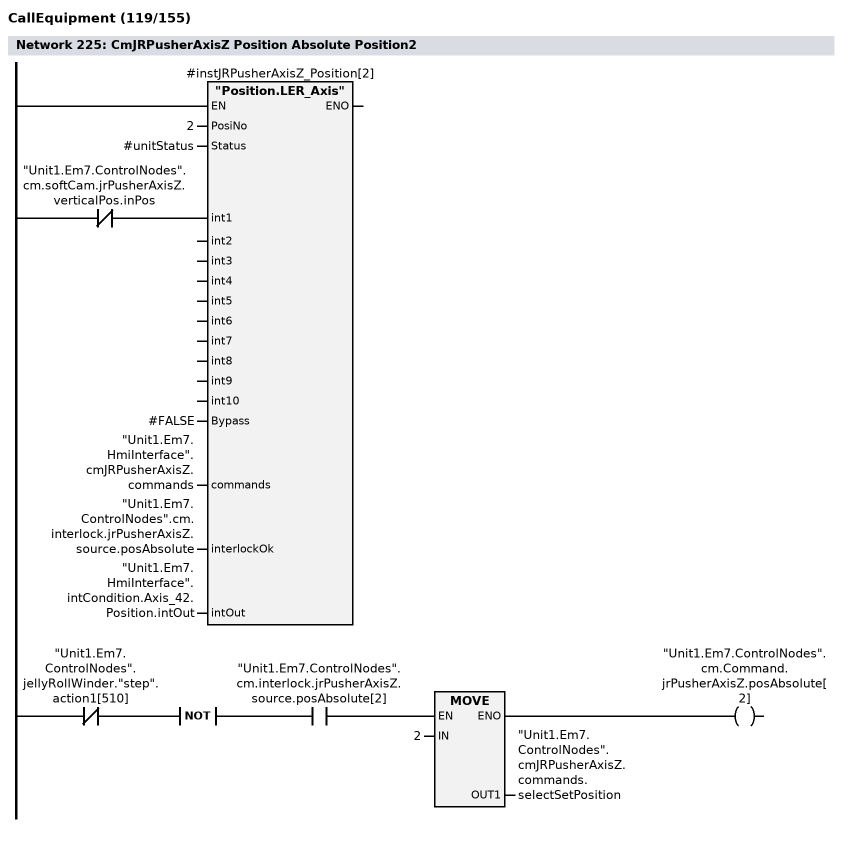
   RUNG wire#powerrail
      #instJRPusherAxisZ_Position[2](int1 := wire#w1, PosiNo := 2, Status := #unitStatus, int2 :=, int3 :=, int4 :=, int5 :=, int6 :=, int7 :=, int8 :=, int9 :=, int10 :=, Bypass := #FALSE, commands := "Unit1.Em7.HmiInterface".cmJRPusherAxisZ.commands, interlockOk := "Unit1.Em7.ControlNodes".cm.interlock.jrPusherAxisZ.source.posAbsolute, intOut := "Unit1.Em7.HmiInterface".intCondition.Axis_42.Position.intOut)
   END_RUNG
   RUNG wire#powerrail
      I_Contact( "Unit1.Em7.ControlNodes".cm.softCam.jrPusherAxisZ.verticalPos.inPos )
   END_RUNG wire#w1
   RUNG wire#powerrail
      I_Contact( "Unit1.Em7.ControlNodes".jellyRollWinder."step".action1[510] )
      Not()
      Contact( "Unit1.Em7.ControlNodes".cm.interlock.jrPusherAxisZ.source.posAbsolute[2] )
      Move(in := 2, out1 => "Unit1.Em7.ControlNodes".cmJRPusherAxisZ.commands.selectSetPosition)
      Coil( "Unit1.Em7.ControlNodes".cm.Command.jrPusherAxisZ.posAbsolute[2] )
   END_RUNG
   // the same network as SCL:
   #instJRPusherAxisZ_Position[2](PosiNo := 2,   // "Position.LER_Axis"
                           Status := #unitStatus,
                           int1 := NOT "Unit1.Em7.ControlNodes".cm.softCam.jrPusherAxisZ.verticalPos.inPos,
                           Bypass := #FALSE,
                           commands := "Unit1.Em7.HmiInterface".cmJRPusherAxisZ.commands,
                           interlockOk := "Unit1.Em7.ControlNodes".cm.interlock.jrPusherAxisZ.source.posAbsolute,
                           intOut := "Unit1.Em7.HmiInterface".intCondition.Axis_42.Position.intOut);
   #_w1 := NOT (NOT "Unit1.Em7.ControlNodes".jellyRollWinder."step".action1[510]) AND "Unit1.Em7.ControlNodes".cm.interlock.jrPusherAxisZ.source.posAbsolute[2];
   IF #_w1 THEN "Unit1.Em7.ControlNodes".cmJRPusherAxisZ.commands.selectSetPosition := 2; END_IF;
   "Unit1.Em7.ControlNodes".cm.Command.jrPusherAxisZ.posAbsolute[2] := #_w1;
END_REGION

REGION Network 226: CmJRPusherAxisZ Position Absolute Position3
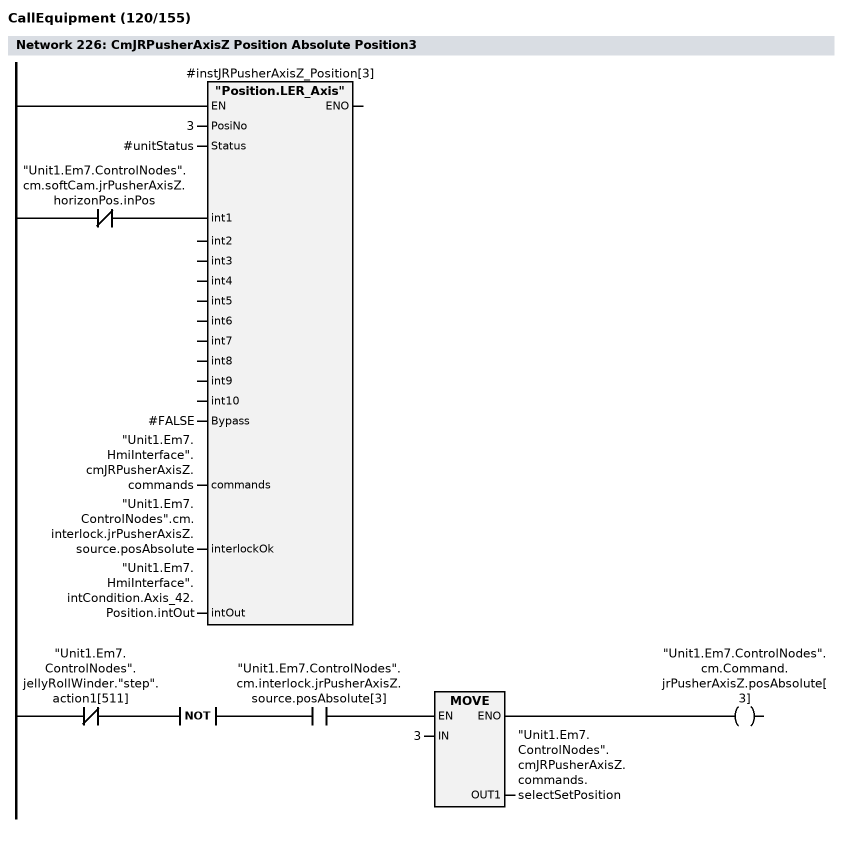
   RUNG wire#powerrail
      #instJRPusherAxisZ_Position[3](int1 := wire#w1, PosiNo := 3, Status := #unitStatus, int2 :=, int3 :=, int4 :=, int5 :=, int6 :=, int7 :=, int8 :=, int9 :=, int10 :=, Bypass := #FALSE, commands := "Unit1.Em7.HmiInterface".cmJRPusherAxisZ.commands, interlockOk := "Unit1.Em7.ControlNodes".cm.interlock.jrPusherAxisZ.source.posAbsolute, intOut := "Unit1.Em7.HmiInterface".intCondition.Axis_42.Position.intOut)
   END_RUNG
   RUNG wire#powerrail
      I_Contact( "Unit1.Em7.ControlNodes".cm.softCam.jrPusherAxisZ.horizonPos.inPos )
   END_RUNG wire#w1
   RUNG wire#powerrail
      I_Contact( "Unit1.Em7.ControlNodes".jellyRollWinder."step".action1[511] )
      Not()
      Contact( "Unit1.Em7.ControlNodes".cm.interlock.jrPusherAxisZ.source.posAbsolute[3] )
      Move(in := 3, out1 => "Unit1.Em7.ControlNodes".cmJRPusherAxisZ.commands.selectSetPosition)
      Coil( "Unit1.Em7.ControlNodes".cm.Command.jrPusherAxisZ.posAbsolute[3] )
   END_RUNG
   // the same network as SCL:
   #instJRPusherAxisZ_Position[3](PosiNo := 3,   // "Position.LER_Axis"
                           Status := #unitStatus,
                           int1 := NOT "Unit1.Em7.ControlNodes".cm.softCam.jrPusherAxisZ.horizonPos.inPos,
                           Bypass := #FALSE,
                           commands := "Unit1.Em7.HmiInterface".cmJRPusherAxisZ.commands,
                           interlockOk := "Unit1.Em7.ControlNodes".cm.interlock.jrPusherAxisZ.source.posAbsolute,
                           intOut := "Unit1.Em7.HmiInterface".intCondition.Axis_42.Position.intOut);
   #_w1 := NOT (NOT "Unit1.Em7.ControlNodes".jellyRollWinder."step".action1[511]) AND "Unit1.Em7.ControlNodes".cm.interlock.jrPusherAxisZ.source.posAbsolute[3];
   IF #_w1 THEN "Unit1.Em7.ControlNodes".cmJRPusherAxisZ.commands.selectSetPosition := 3; END_IF;
   "Unit1.Em7.ControlNodes".cm.Command.jrPusherAxisZ.posAbsolute[3] := #_w1;
END_REGION

REGION Network 227: CmJRPusherAxisZ Position Absolute Position4
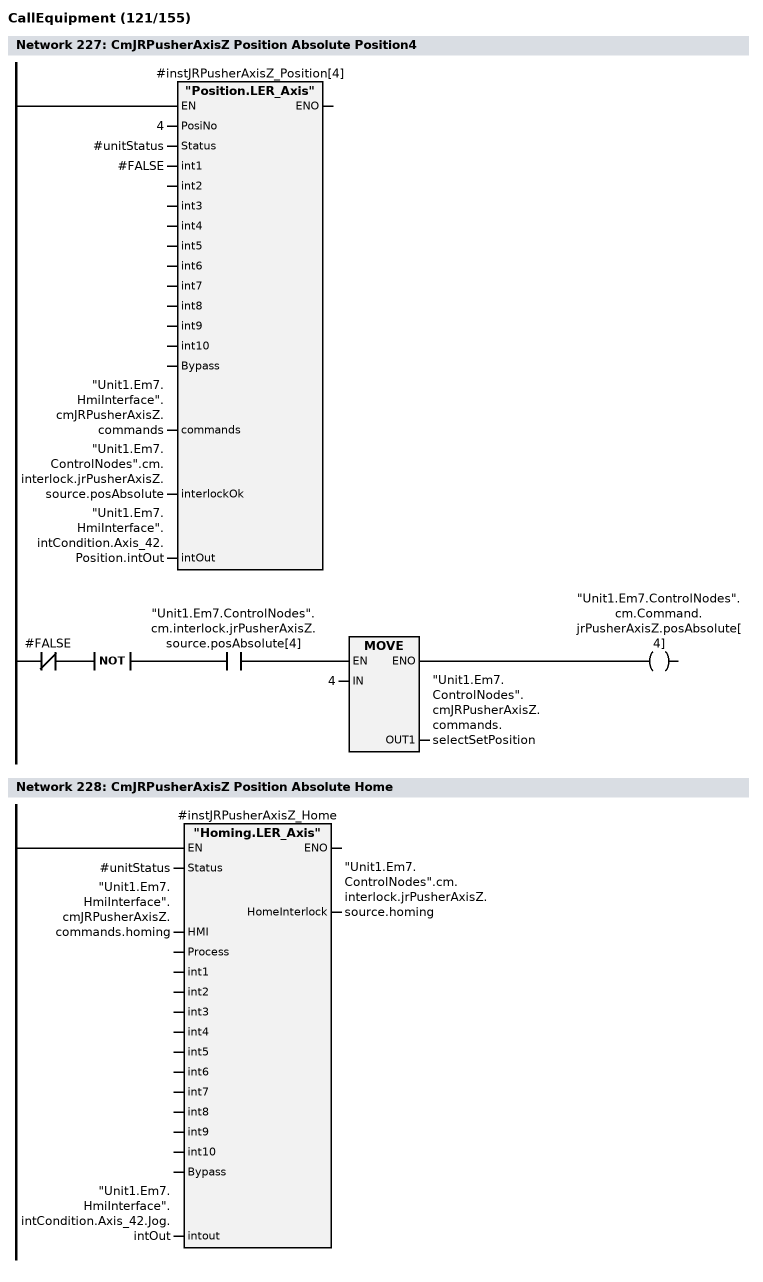
   RUNG wire#powerrail
      #instJRPusherAxisZ_Position[4](PosiNo := 4, Status := #unitStatus, int1 := #FALSE, int2 :=, int3 :=, int4 :=, int5 :=, int6 :=, int7 :=, int8 :=, int9 :=, int10 :=, Bypass :=, commands := "Unit1.Em7.HmiInterface".cmJRPusherAxisZ.commands, interlockOk := "Unit1.Em7.ControlNodes".cm.interlock.jrPusherAxisZ.source.posAbsolute, intOut := "Unit1.Em7.HmiInterface".intCondition.Axis_42.Position.intOut)
   END_RUNG
   RUNG wire#powerrail
      I_Contact( #FALSE )
      Not()
      Contact( "Unit1.Em7.ControlNodes".cm.interlock.jrPusherAxisZ.source.posAbsolute[4] )
      Move(in := 4, out1 => "Unit1.Em7.ControlNodes".cmJRPusherAxisZ.commands.selectSetPosition)
      Coil( "Unit1.Em7.ControlNodes".cm.Command.jrPusherAxisZ.posAbsolute[4] )
   END_RUNG
   // the same network as SCL:
   #instJRPusherAxisZ_Position[4](PosiNo := 4,   // "Position.LER_Axis"
                           Status := #unitStatus,
                           int1 := #FALSE,
                           commands := "Unit1.Em7.HmiInterface".cmJRPusherAxisZ.commands,
                           interlockOk := "Unit1.Em7.ControlNodes".cm.interlock.jrPusherAxisZ.source.posAbsolute,
                           intOut := "Unit1.Em7.HmiInterface".intCondition.Axis_42.Position.intOut);
   #_w1 := NOT (NOT #FALSE) AND "Unit1.Em7.ControlNodes".cm.interlock.jrPusherAxisZ.source.posAbsolute[4];
   IF #_w1 THEN "Unit1.Em7.ControlNodes".cmJRPusherAxisZ.commands.selectSetPosition := 4; END_IF;
   "Unit1.Em7.ControlNodes".cm.Command.jrPusherAxisZ.posAbsolute[4] := #_w1;
END_REGION

REGION Network 228: CmJRPusherAxisZ Position Absolute Home
   RUNG wire#powerrail
      #instJRPusherAxisZ_Home(Status := #unitStatus, HMI := "Unit1.Em7.HmiInterface".cmJRPusherAxisZ.commands.homing, Process :=, int1 :=, int2 :=, int3 :=, int4 :=, int5 :=, int6 :=, int7 :=, int8 :=, int9 :=, int10 :=, Bypass :=, intout := "Unit1.Em7.HmiInterface".intCondition.Axis_42.Jog.intOut, HomeInterlock => "Unit1.Em7.ControlNodes".cm.interlock.jrPusherAxisZ.source.homing)
   END_RUNG
   // the same network as SCL:
   #instJRPusherAxisZ_Home(Status := #unitStatus,   // "Homing.LER_Axis"
                           HMI := "Unit1.Em7.HmiInterface".cmJRPusherAxisZ.commands.homing,
                           intout := "Unit1.Em7.HmiInterface".intCondition.Axis_42.Jog.intOut,
                           HomeInterlock => "Unit1.Em7.ControlNodes".cm.interlock.jrPusherAxisZ.source.homing);
END_REGION

REGION Network 229: CmJRPusherAxisZ Position Absolute Position5
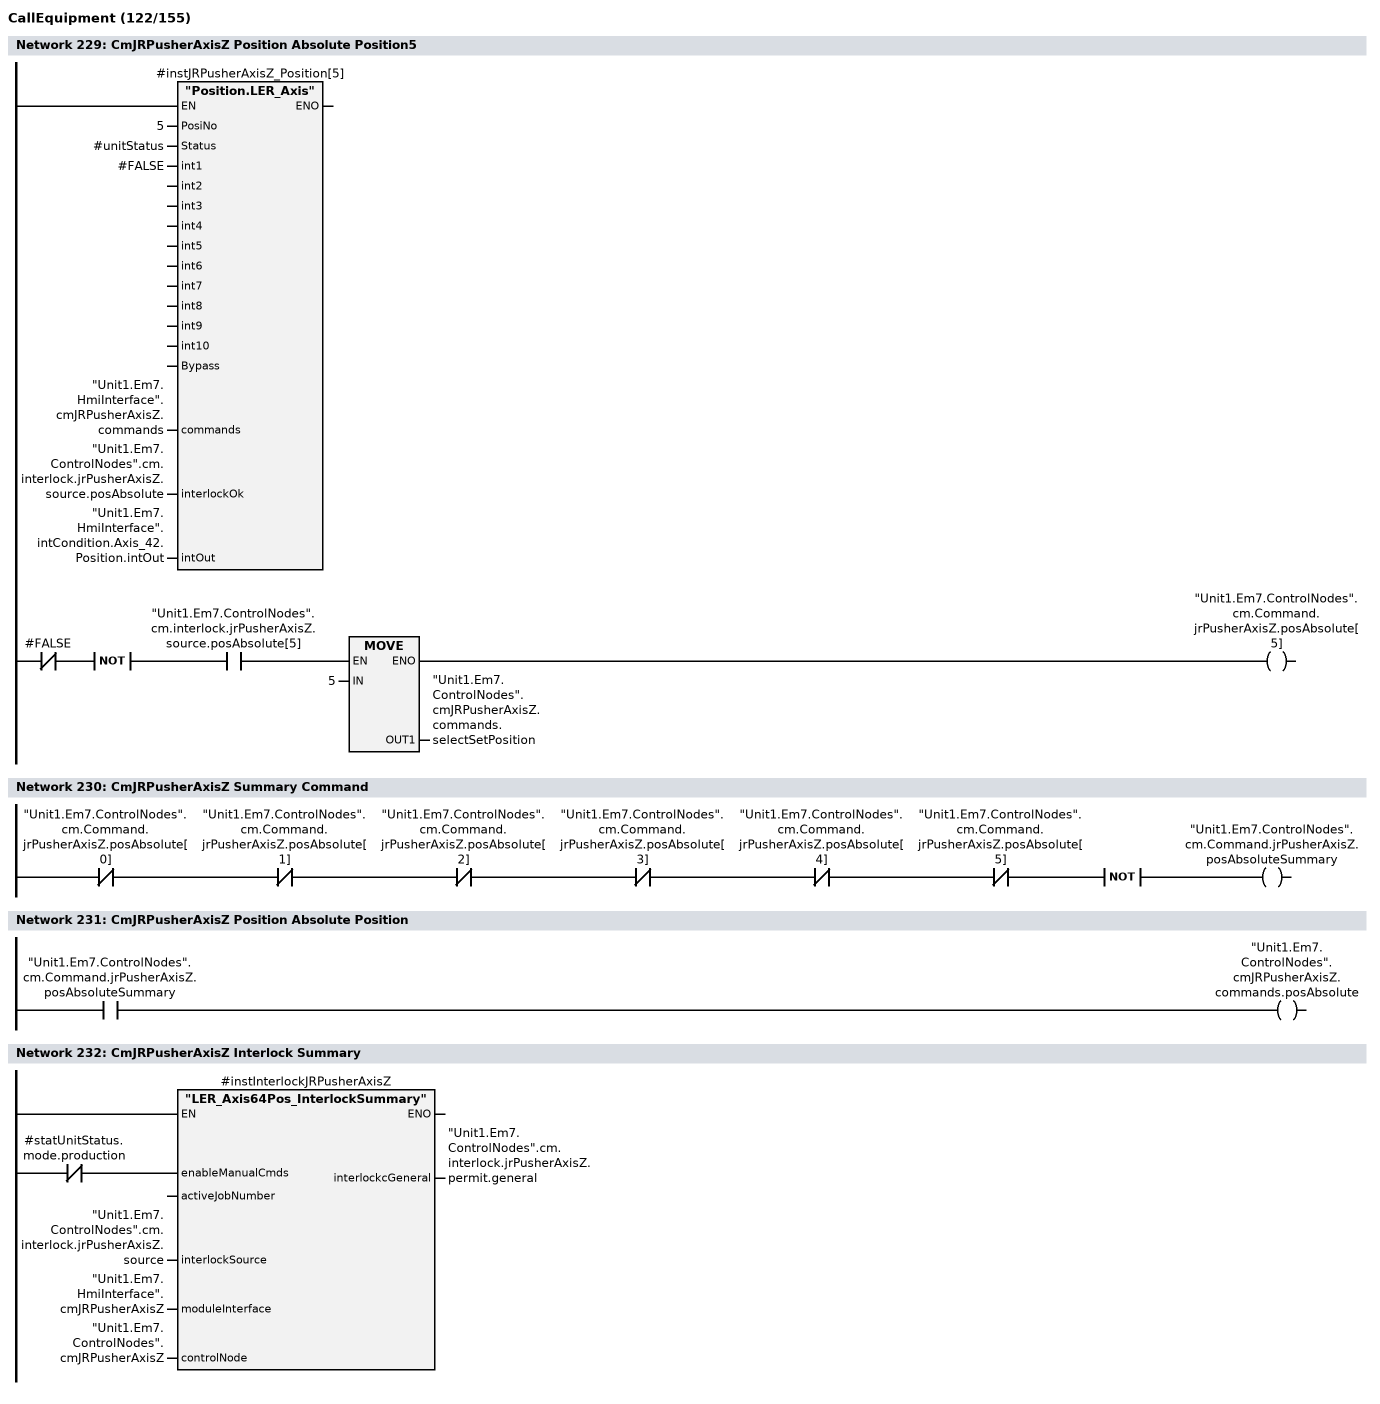
   RUNG wire#powerrail
      #instJRPusherAxisZ_Position[5](PosiNo := 5, Status := #unitStatus, int1 := #FALSE, int2 :=, int3 :=, int4 :=, int5 :=, int6 :=, int7 :=, int8 :=, int9 :=, int10 :=, Bypass :=, commands := "Unit1.Em7.HmiInterface".cmJRPusherAxisZ.commands, interlockOk := "Unit1.Em7.ControlNodes".cm.interlock.jrPusherAxisZ.source.posAbsolute, intOut := "Unit1.Em7.HmiInterface".intCondition.Axis_42.Position.intOut)
   END_RUNG
   RUNG wire#powerrail
      I_Contact( #FALSE )
      Not()
      Contact( "Unit1.Em7.ControlNodes".cm.interlock.jrPusherAxisZ.source.posAbsolute[5] )
      Move(in := 5, out1 => "Unit1.Em7.ControlNodes".cmJRPusherAxisZ.commands.selectSetPosition)
      Coil( "Unit1.Em7.ControlNodes".cm.Command.jrPusherAxisZ.posAbsolute[5] )
   END_RUNG
   // the same network as SCL:
   #instJRPusherAxisZ_Position[5](PosiNo := 5,   // "Position.LER_Axis"
                           Status := #unitStatus,
                           int1 := #FALSE,
                           commands := "Unit1.Em7.HmiInterface".cmJRPusherAxisZ.commands,
                           interlockOk := "Unit1.Em7.ControlNodes".cm.interlock.jrPusherAxisZ.source.posAbsolute,
                           intOut := "Unit1.Em7.HmiInterface".intCondition.Axis_42.Position.intOut);
   #_w1 := NOT (NOT #FALSE) AND "Unit1.Em7.ControlNodes".cm.interlock.jrPusherAxisZ.source.posAbsolute[5];
   IF #_w1 THEN "Unit1.Em7.ControlNodes".cmJRPusherAxisZ.commands.selectSetPosition := 5; END_IF;
   "Unit1.Em7.ControlNodes".cm.Command.jrPusherAxisZ.posAbsolute[5] := #_w1;
END_REGION

REGION Network 230: CmJRPusherAxisZ Summary Command
   RUNG wire#powerrail
      I_Contact( "Unit1.Em7.ControlNodes".cm.Command.jrPusherAxisZ.posAbsolute[0] )
      I_Contact( "Unit1.Em7.ControlNodes".cm.Command.jrPusherAxisZ.posAbsolute[1] )
      I_Contact( "Unit1.Em7.ControlNodes".cm.Command.jrPusherAxisZ.posAbsolute[2] )
      I_Contact( "Unit1.Em7.ControlNodes".cm.Command.jrPusherAxisZ.posAbsolute[3] )
      I_Contact( "Unit1.Em7.ControlNodes".cm.Command.jrPusherAxisZ.posAbsolute[4] )
      I_Contact( "Unit1.Em7.ControlNodes".cm.Command.jrPusherAxisZ.posAbsolute[5] )
      Not()
      Coil( "Unit1.Em7.ControlNodes".cm.Command.jrPusherAxisZ.posAbsoluteSummary )
   END_RUNG
   // the same network as SCL:
   "Unit1.Em7.ControlNodes".cm.Command.jrPusherAxisZ.posAbsoluteSummary := NOT (NOT "Unit1.Em7.ControlNodes".cm.Command.jrPusherAxisZ.posAbsolute[0] AND NOT "Unit1.Em7.ControlNodes".cm.Command.jrPusherAxisZ.posAbsolute[1] AND NOT "Unit1.Em7.ControlNodes".cm.Command.jrPusherAxisZ.posAbsolute[2] AND NOT "Unit1.Em7.ControlNodes".cm.Command.jrPusherAxisZ.posAbsolute[3] AND NOT "Unit1.Em7.ControlNodes".cm.Command.jrPusherAxisZ.posAbsolute[4] AND NOT "Unit1.Em7.ControlNodes".cm.Command.jrPusherAxisZ.posAbsolute[5]);
END_REGION

REGION Network 231: CmJRPusherAxisZ Position Absolute Position
   RUNG wire#powerrail
      Contact( "Unit1.Em7.ControlNodes".cm.Command.jrPusherAxisZ.posAbsoluteSummary )
      Coil( "Unit1.Em7.ControlNodes".cmJRPusherAxisZ.commands.posAbsolute )
   END_RUNG
   // the same network as SCL:
   "Unit1.Em7.ControlNodes".cmJRPusherAxisZ.commands.posAbsolute := "Unit1.Em7.ControlNodes".cm.Command.jrPusherAxisZ.posAbsoluteSummary;
END_REGION

REGION Network 232: CmJRPusherAxisZ Interlock Summary
   RUNG wire#powerrail
      #instInterlockJRPusherAxisZ(enableManualCmds := wire#w1, activeJobNumber :=, interlockSource := "Unit1.Em7.ControlNodes".cm.interlock.jrPusherAxisZ.source, moduleInterface := "Unit1.Em7.HmiInterface".cmJRPusherAxisZ, controlNode := "Unit1.Em7.ControlNodes".cmJRPusherAxisZ, interlockcGeneral => "Unit1.Em7.ControlNodes".cm.interlock.jrPusherAxisZ.permit.general)
   END_RUNG
   RUNG wire#powerrail
      I_Contact( #statUnitStatus.mode.production )
   END_RUNG wire#w1
   // the same network as SCL:
   #instInterlockJRPusherAxisZ(enableManualCmds := NOT #statUnitStatus.mode.production,   // "LER_Axis64Pos_InterlockSummary"
                           interlockSource := "Unit1.Em7.ControlNodes".cm.interlock.jrPusherAxisZ.source,
                           moduleInterface := "Unit1.Em7.HmiInterface".cmJRPusherAxisZ,
                           controlNode := "Unit1.Em7.ControlNodes".cmJRPusherAxisZ,
                           interlockcGeneral => "Unit1.Em7.ControlNodes".cm.interlock.jrPusherAxisZ.permit.general);
END_REGION

REGION Network 233: CmJRPusherAxisZ velocity/speed
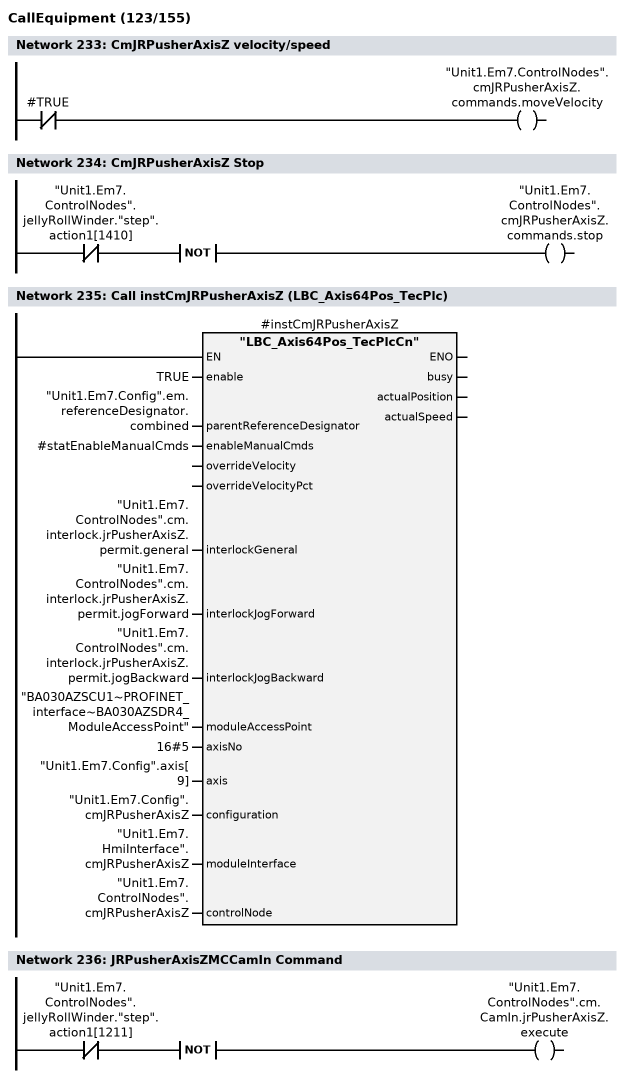
   RUNG wire#powerrail
      I_Contact( #TRUE )
      Coil( "Unit1.Em7.ControlNodes".cmJRPusherAxisZ.commands.moveVelocity )
   END_RUNG
   // the same network as SCL:
   "Unit1.Em7.ControlNodes".cmJRPusherAxisZ.commands.moveVelocity := NOT #TRUE;
END_REGION

REGION Network 234: CmJRPusherAxisZ Stop
   RUNG wire#powerrail
      I_Contact( "Unit1.Em7.ControlNodes".jellyRollWinder."step".action1[1410] )
      Not()
      Coil( "Unit1.Em7.ControlNodes".cmJRPusherAxisZ.commands.stop )
   END_RUNG
   // the same network as SCL:
   "Unit1.Em7.ControlNodes".cmJRPusherAxisZ.commands.stop := NOT (NOT "Unit1.Em7.ControlNodes".jellyRollWinder."step".action1[1410]);
END_REGION

REGION Network 235: Call instCmJRPusherAxisZ (LBC_Axis64Pos_TecPlc)
   RUNG wire#powerrail
      #instCmJRPusherAxisZ(enable := TRUE, parentReferenceDesignator := "Unit1.Em7.Config".em.referenceDesignator.combined, enableManualCmds := #statEnableManualCmds, overrideVelocity :=, overrideVelocityPct :=, interlockGeneral := "Unit1.Em7.ControlNodes".cm.interlock.jrPusherAxisZ.permit.general, interlockJogForward := "Unit1.Em7.ControlNodes".cm.interlock.jrPusherAxisZ.permit.jogForward, interlockJogBackward := "Unit1.Em7.ControlNodes".cm.interlock.jrPusherAxisZ.permit.jogBackward, moduleAccessPoint := "BA030AZSCU1~PROFINET_interface~BA030AZSDR4_ModuleAccessPoint", axisNo := 16#5, axis := "Unit1.Em7.Config".axis[9], configuration := "Unit1.Em7.Config".cmJRPusherAxisZ, moduleInterface := "Unit1.Em7.HmiInterface".cmJRPusherAxisZ, controlNode := "Unit1.Em7.ControlNodes".cmJRPusherAxisZ, busy =>, actualPosition =>, actualSpeed =>)
   END_RUNG
   // the same network as SCL:
   #instCmJRPusherAxisZ(enable := TRUE,   // "LBC_Axis64Pos_TecPlcCn"
                        parentReferenceDesignator := "Unit1.Em7.Config".em.referenceDesignator.combined,
                        enableManualCmds := #statEnableManualCmds,
                        interlockGeneral := "Unit1.Em7.ControlNodes".cm.interlock.jrPusherAxisZ.permit.general,
                        interlockJogForward := "Unit1.Em7.ControlNodes".cm.interlock.jrPusherAxisZ.permit.jogForward,
                        interlockJogBackward := "Unit1.Em7.ControlNodes".cm.interlock.jrPusherAxisZ.permit.jogBackward,
                        moduleAccessPoint := "BA030AZSCU1~PROFINET_interface~BA030AZSDR4_ModuleAccessPoint",
                        axisNo := 16#5,
                        axis := "Unit1.Em7.Config".axis[9],
                        configuration := "Unit1.Em7.Config".cmJRPusherAxisZ,
                        moduleInterface := "Unit1.Em7.HmiInterface".cmJRPusherAxisZ,
                        controlNode := "Unit1.Em7.ControlNodes".cmJRPusherAxisZ);
END_REGION

REGION Network 236: JRPusherAxisZMCCamIn Command
   RUNG wire#powerrail
      I_Contact( "Unit1.Em7.ControlNodes".jellyRollWinder."step".action1[1211] )
      Not()
      Coil( "Unit1.Em7.ControlNodes".cm.CamIn.jrPusherAxisZ.execute )
   END_RUNG
   // the same network as SCL:
   "Unit1.Em7.ControlNodes".cm.CamIn.jrPusherAxisZ.execute := NOT (NOT "Unit1.Em7.ControlNodes".jellyRollWinder."step".action1[1211]);
END_REGION

REGION Network 237: Call instJRPusherAxisZMCCamIn
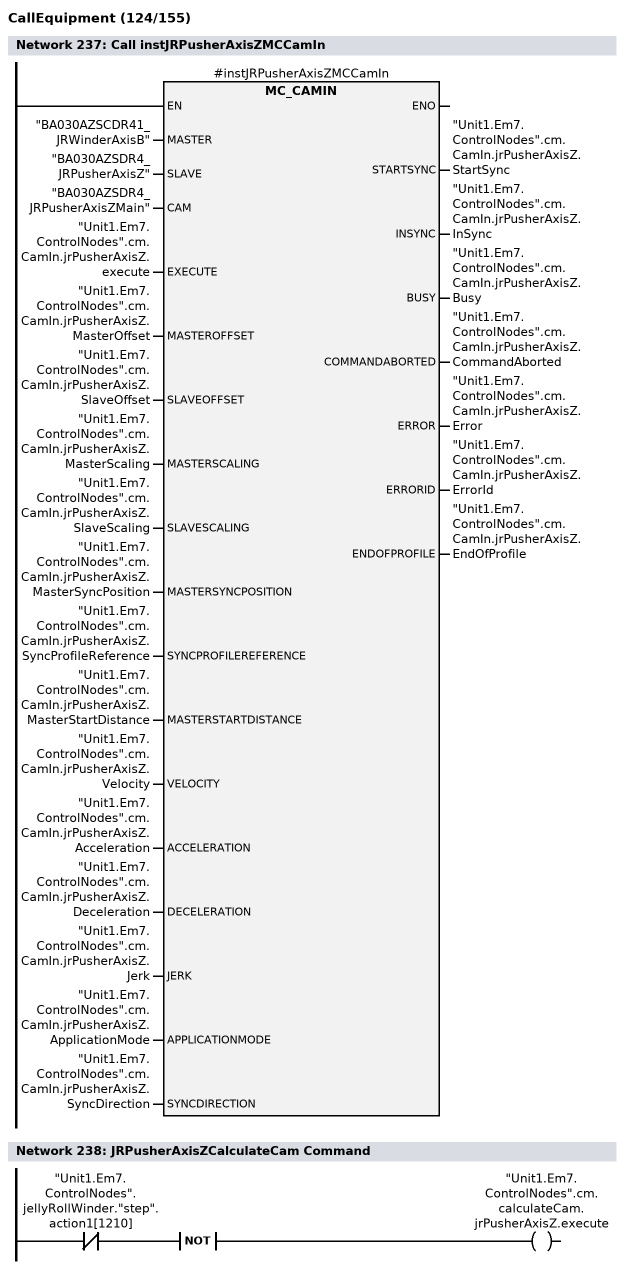
   RUNG wire#powerrail
      #instJRPusherAxisZMCCamIn.MC_CAMIN(Master := "BA030AZSCDR41_JRWinderAxisB", Slave := "BA030AZSDR4_JRPusherAxisZ", Cam := "BA030AZSDR4_JRPusherAxisZMain", Execute := "Unit1.Em7.ControlNodes".cm.CamIn.jrPusherAxisZ.execute, MasterOffset := "Unit1.Em7.ControlNodes".cm.CamIn.jrPusherAxisZ.MasterOffset, SlaveOffset := "Unit1.Em7.ControlNodes".cm.CamIn.jrPusherAxisZ.SlaveOffset, MasterScaling := "Unit1.Em7.ControlNodes".cm.CamIn.jrPusherAxisZ.MasterScaling, SlaveScaling := "Unit1.Em7.ControlNodes".cm.CamIn.jrPusherAxisZ.SlaveScaling, MasterSyncPosition := "Unit1.Em7.ControlNodes".cm.CamIn.jrPusherAxisZ.MasterSyncPosition, SyncProfileReference := "Unit1.Em7.ControlNodes".cm.CamIn.jrPusherAxisZ.SyncProfileReference, MasterStartDistance := "Unit1.Em7.ControlNodes".cm.CamIn.jrPusherAxisZ.MasterStartDistance, Velocity := "Unit1.Em7.ControlNodes".cm.CamIn.jrPusherAxisZ.Velocity, Acceleration := "Unit1.Em7.ControlNodes".cm.CamIn.jrPusherAxisZ.Acceleration, Deceleration := "Unit1.Em7.ControlNodes".cm.CamIn.jrPusherAxisZ.Deceleration, Jerk := "Unit1.Em7.ControlNodes".cm.CamIn.jrPusherAxisZ.Jerk, ApplicationMode := "Unit1.Em7.ControlNodes".cm.CamIn.jrPusherAxisZ.ApplicationMode, SyncDirection := "Unit1.Em7.ControlNodes".cm.CamIn.jrPusherAxisZ.SyncDirection, StartSync => "Unit1.Em7.ControlNodes".cm.CamIn.jrPusherAxisZ.StartSync, InSync => "Unit1.Em7.ControlNodes".cm.CamIn.jrPusherAxisZ.InSync, Busy => "Unit1.Em7.ControlNodes".cm.CamIn.jrPusherAxisZ.Busy, CommandAborted => "Unit1.Em7.ControlNodes".cm.CamIn.jrPusherAxisZ.CommandAborted, Error => "Unit1.Em7.ControlNodes".cm.CamIn.jrPusherAxisZ.Error, ErrorId => "Unit1.Em7.ControlNodes".cm.CamIn.jrPusherAxisZ.ErrorId, EndOfProfile => "Unit1.Em7.ControlNodes".cm.CamIn.jrPusherAxisZ.EndOfProfile)
   END_RUNG
   // the same network as SCL:
   #instJRPusherAxisZMCCamIn(Master := "BA030AZSCDR41_JRWinderAxisB",   // MC_CAMIN
                           Slave := "BA030AZSDR4_JRPusherAxisZ",
                           Cam := "BA030AZSDR4_JRPusherAxisZMain",
                           Execute := "Unit1.Em7.ControlNodes".cm.CamIn.jrPusherAxisZ.execute,
                           MasterOffset := "Unit1.Em7.ControlNodes".cm.CamIn.jrPusherAxisZ.MasterOffset,
                           SlaveOffset := "Unit1.Em7.ControlNodes".cm.CamIn.jrPusherAxisZ.SlaveOffset,
                           MasterScaling := "Unit1.Em7.ControlNodes".cm.CamIn.jrPusherAxisZ.MasterScaling,
                           SlaveScaling := "Unit1.Em7.ControlNodes".cm.CamIn.jrPusherAxisZ.SlaveScaling,
                           MasterSyncPosition := "Unit1.Em7.ControlNodes".cm.CamIn.jrPusherAxisZ.MasterSyncPosition,
                           SyncProfileReference := "Unit1.Em7.ControlNodes".cm.CamIn.jrPusherAxisZ.SyncProfileReference,
                           MasterStartDistance := "Unit1.Em7.ControlNodes".cm.CamIn.jrPusherAxisZ.MasterStartDistance,
                           Velocity := "Unit1.Em7.ControlNodes".cm.CamIn.jrPusherAxisZ.Velocity,
                           Acceleration := "Unit1.Em7.ControlNodes".cm.CamIn.jrPusherAxisZ.Acceleration,
                           Deceleration := "Unit1.Em7.ControlNodes".cm.CamIn.jrPusherAxisZ.Deceleration,
                           Jerk := "Unit1.Em7.ControlNodes".cm.CamIn.jrPusherAxisZ.Jerk,
                           ApplicationMode := "Unit1.Em7.ControlNodes".cm.CamIn.jrPusherAxisZ.ApplicationMode,
                           SyncDirection := "Unit1.Em7.ControlNodes".cm.CamIn.jrPusherAxisZ.SyncDirection,
                           StartSync => "Unit1.Em7.ControlNodes".cm.CamIn.jrPusherAxisZ.StartSync,
                           InSync => "Unit1.Em7.ControlNodes".cm.CamIn.jrPusherAxisZ.InSync,
                           Busy => "Unit1.Em7.ControlNodes".cm.CamIn.jrPusherAxisZ.Busy,
                           CommandAborted => "Unit1.Em7.ControlNodes".cm.CamIn.jrPusherAxisZ.CommandAborted,
                           Error => "Unit1.Em7.ControlNodes".cm.CamIn.jrPusherAxisZ.Error,
                           ErrorId => "Unit1.Em7.ControlNodes".cm.CamIn.jrPusherAxisZ.ErrorId,
                           EndOfProfile => "Unit1.Em7.ControlNodes".cm.CamIn.jrPusherAxisZ.EndOfProfile);
END_REGION

REGION Network 238: JRPusherAxisZCalculateCam Command
   RUNG wire#powerrail
      I_Contact( "Unit1.Em7.ControlNodes".jellyRollWinder."step".action1[1210] )
      Not()
      Coil( "Unit1.Em7.ControlNodes".cm.calculateCam.jrPusherAxisZ.execute )
   END_RUNG
   // the same network as SCL:
   "Unit1.Em7.ControlNodes".cm.calculateCam.jrPusherAxisZ.execute := NOT (NOT "Unit1.Em7.ControlNodes".jellyRollWinder."step".action1[1210]);
END_REGION

REGION Network 239: Call instJRPusherAxisZCalculateCam
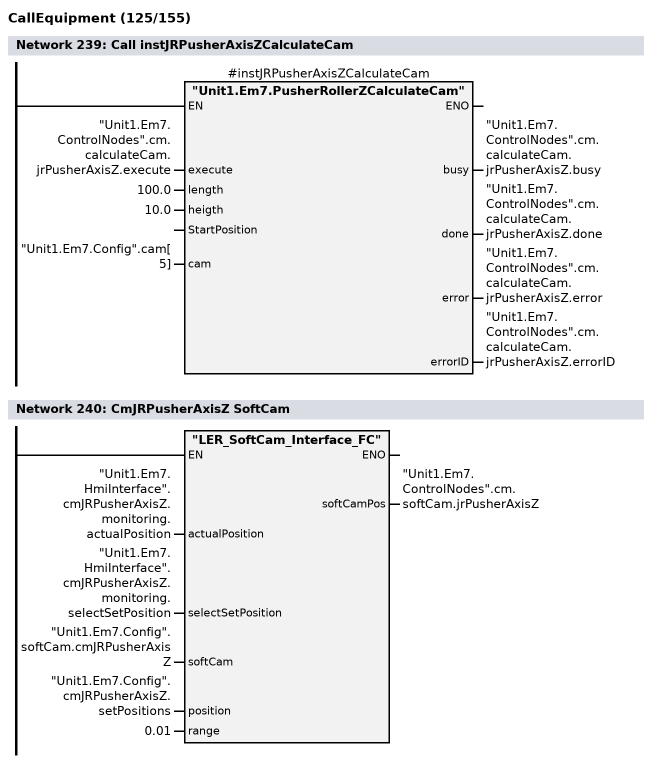
   RUNG wire#powerrail
      #instJRPusherAxisZCalculateCam(execute := "Unit1.Em7.ControlNodes".cm.calculateCam.jrPusherAxisZ.execute, length := 100.0, heigth := 10.0, StartPosition :=, cam := "Unit1.Em7.Config".cam[5], busy => "Unit1.Em7.ControlNodes".cm.calculateCam.jrPusherAxisZ.busy, done => "Unit1.Em7.ControlNodes".cm.calculateCam.jrPusherAxisZ.done, error => "Unit1.Em7.ControlNodes".cm.calculateCam.jrPusherAxisZ.error, errorID => "Unit1.Em7.ControlNodes".cm.calculateCam.jrPusherAxisZ.errorID)
   END_RUNG
   // the same network as SCL:
   #instJRPusherAxisZCalculateCam(execute := "Unit1.Em7.ControlNodes".cm.calculateCam.jrPusherAxisZ.execute,   // "Unit1.Em7.PusherRollerZCalculateCam"
                           length := 100.0,
                           heigth := 10.0,
                           cam := "Unit1.Em7.Config".cam[5],
                           busy => "Unit1.Em7.ControlNodes".cm.calculateCam.jrPusherAxisZ.busy,
                           done => "Unit1.Em7.ControlNodes".cm.calculateCam.jrPusherAxisZ.done,
                           error => "Unit1.Em7.ControlNodes".cm.calculateCam.jrPusherAxisZ.error,
                           errorID => "Unit1.Em7.ControlNodes".cm.calculateCam.jrPusherAxisZ.errorID);
END_REGION

REGION Network 240: CmJRPusherAxisZ SoftCam
   RUNG wire#powerrail
      "LER_SoftCam_Interface_FC"(actualPosition := "Unit1.Em7.HmiInterface".cmJRPusherAxisZ.monitoring.actualPosition, selectSetPosition := "Unit1.Em7.HmiInterface".cmJRPusherAxisZ.monitoring.selectSetPosition, softCam := "Unit1.Em7.Config".softCam.cmJRPusherAxisZ, position := "Unit1.Em7.Config".cmJRPusherAxisZ.setPositions, range := 0.01, softCamPos => "Unit1.Em7.ControlNodes".cm.softCam.jrPusherAxisZ)
   END_RUNG
   // the same network as SCL:
   "LER_SoftCam_Interface_FC"(actualPosition := "Unit1.Em7.HmiInterface".cmJRPusherAxisZ.monitoring.actualPosition,
                           selectSetPosition := "Unit1.Em7.HmiInterface".cmJRPusherAxisZ.monitoring.selectSetPosition,
                           softCam := "Unit1.Em7.Config".softCam.cmJRPusherAxisZ,
                           position := "Unit1.Em7.Config".cmJRPusherAxisZ.setPositions,
                           range := 0.01,
                           softCamPos => "Unit1.Em7.ControlNodes".cm.softCam.jrPusherAxisZ);
END_REGION

REGION Network 241: ******************** Brake Test (Axis) ********************
END_REGION

REGION Network 242: Sepa Clamp And Cutter Z-Axis Brake Test
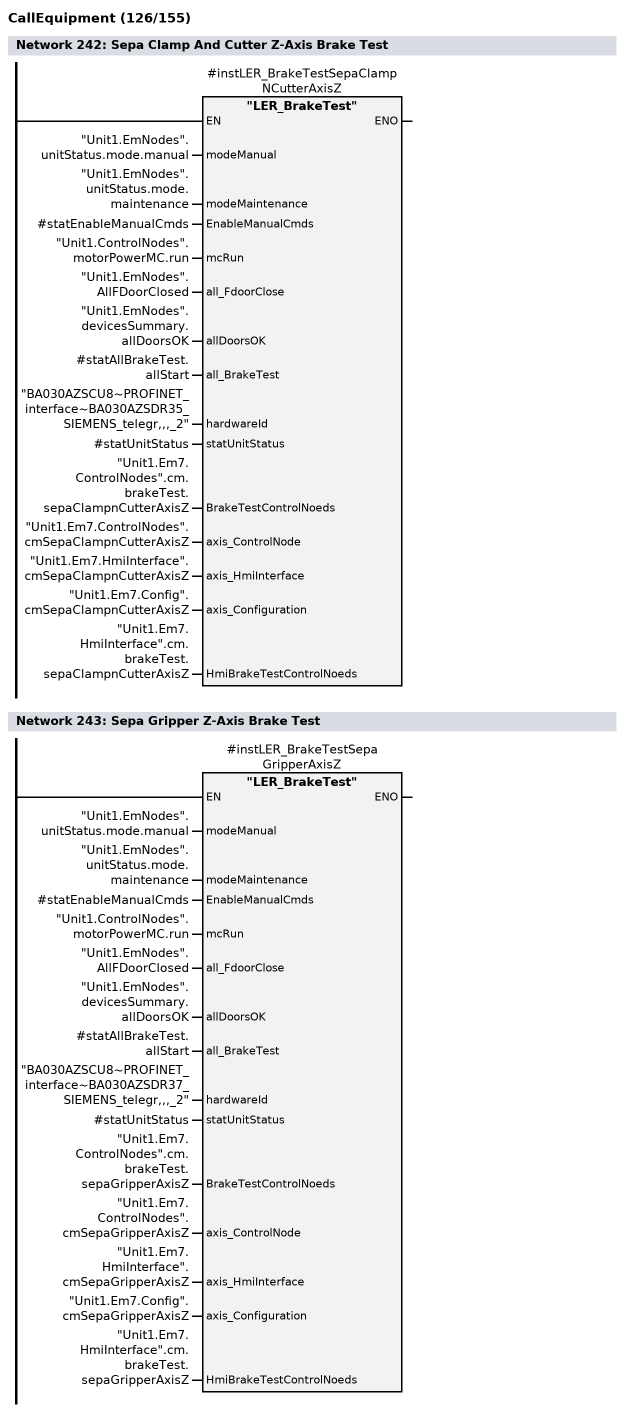
   RUNG wire#powerrail
      #instLER_BrakeTestSepaClampNCutterAxisZ(modeManual := "Unit1.EmNodes".unitStatus.mode.manual, modeMaintenance := "Unit1.EmNodes".unitStatus.mode.maintenance, EnableManualCmds := #statEnableManualCmds, mcRun := "Unit1.ControlNodes".motorPowerMC.run, all_FdoorClose := "Unit1.EmNodes".AllFDoorClosed, allDoorsOK := "Unit1.EmNodes".devicesSummary.allDoorsOK, all_BrakeTest := #statAllBrakeTest.allStart, hardwareId := "BA030AZSCU8~PROFINET_interface~BA030AZSDR35_SIEMENS_telegr,,,_2", statUnitStatus := #statUnitStatus, BrakeTestControlNoeds := "Unit1.Em7.ControlNodes".cm.brakeTest.sepaClampnCutterAxisZ, axis_ControlNode := "Unit1.Em7.ControlNodes".cmSepaClampnCutterAxisZ, axis_HmiInterface := "Unit1.Em7.HmiInterface".cmSepaClampnCutterAxisZ, axis_Configuration := "Unit1.Em7.Config".cmSepaClampnCutterAxisZ, HmiBrakeTestControlNoeds := "Unit1.Em7.HmiInterface".cm.brakeTest.sepaClampnCutterAxisZ)
   END_RUNG
   // the same network as SCL:
   #instLER_BrakeTestSepaClampNCutterAxisZ(modeManual := "Unit1.EmNodes".unitStatus.mode.manual,   // "LER_BrakeTest"
                           modeMaintenance := "Unit1.EmNodes".unitStatus.mode.maintenance,
                           EnableManualCmds := #statEnableManualCmds,
                           mcRun := "Unit1.ControlNodes".motorPowerMC.run,
                           all_FdoorClose := "Unit1.EmNodes".AllFDoorClosed,
                           allDoorsOK := "Unit1.EmNodes".devicesSummary.allDoorsOK,
                           all_BrakeTest := #statAllBrakeTest.allStart,
                           hardwareId := "BA030AZSCU8~PROFINET_interface~BA030AZSDR35_SIEMENS_telegr,,,_2",
                           statUnitStatus := #statUnitStatus,
                           BrakeTestControlNoeds := "Unit1.Em7.ControlNodes".cm.brakeTest.sepaClampnCutterAxisZ,
                           axis_ControlNode := "Unit1.Em7.ControlNodes".cmSepaClampnCutterAxisZ,
                           axis_HmiInterface := "Unit1.Em7.HmiInterface".cmSepaClampnCutterAxisZ,
                           axis_Configuration := "Unit1.Em7.Config".cmSepaClampnCutterAxisZ,
                           HmiBrakeTestControlNoeds := "Unit1.Em7.HmiInterface".cm.brakeTest.sepaClampnCutterAxisZ);
END_REGION

REGION Network 243: Sepa Gripper Z-Axis Brake Test
   RUNG wire#powerrail
      #instLER_BrakeTestSepaGripperAxisZ(modeManual := "Unit1.EmNodes".unitStatus.mode.manual, modeMaintenance := "Unit1.EmNodes".unitStatus.mode.maintenance, EnableManualCmds := #statEnableManualCmds, mcRun := "Unit1.ControlNodes".motorPowerMC.run, all_FdoorClose := "Unit1.EmNodes".AllFDoorClosed, allDoorsOK := "Unit1.EmNodes".devicesSummary.allDoorsOK, all_BrakeTest := #statAllBrakeTest.allStart, hardwareId := "BA030AZSCU8~PROFINET_interface~BA030AZSDR37_SIEMENS_telegr,,,_2", statUnitStatus := #statUnitStatus, BrakeTestControlNoeds := "Unit1.Em7.ControlNodes".cm.brakeTest.sepaGripperAxisZ, axis_ControlNode := "Unit1.Em7.ControlNodes".cmSepaGripperAxisZ, axis_HmiInterface := "Unit1.Em7.HmiInterface".cmSepaGripperAxisZ, axis_Configuration := "Unit1.Em7.Config".cmSepaGripperAxisZ, HmiBrakeTestControlNoeds := "Unit1.Em7.HmiInterface".cm.brakeTest.sepaGripperAxisZ)
   END_RUNG
   // the same network as SCL:
   #instLER_BrakeTestSepaGripperAxisZ(modeManual := "Unit1.EmNodes".unitStatus.mode.manual,   // "LER_BrakeTest"
                           modeMaintenance := "Unit1.EmNodes".unitStatus.mode.maintenance,
                           EnableManualCmds := #statEnableManualCmds,
                           mcRun := "Unit1.ControlNodes".motorPowerMC.run,
                           all_FdoorClose := "Unit1.EmNodes".AllFDoorClosed,
                           allDoorsOK := "Unit1.EmNodes".devicesSummary.allDoorsOK,
                           all_BrakeTest := #statAllBrakeTest.allStart,
                           hardwareId := "BA030AZSCU8~PROFINET_interface~BA030AZSDR37_SIEMENS_telegr,,,_2",
                           statUnitStatus := #statUnitStatus,
                           BrakeTestControlNoeds := "Unit1.Em7.ControlNodes".cm.brakeTest.sepaGripperAxisZ,
                           axis_ControlNode := "Unit1.Em7.ControlNodes".cmSepaGripperAxisZ,
                           axis_HmiInterface := "Unit1.Em7.HmiInterface".cmSepaGripperAxisZ,
                           axis_Configuration := "Unit1.Em7.Config".cmSepaGripperAxisZ,
                           HmiBrakeTestControlNoeds := "Unit1.Em7.HmiInterface".cm.brakeTest.sepaGripperAxisZ);
END_REGION

REGION Network 244: JR Pusher Z-Axis Brake Test
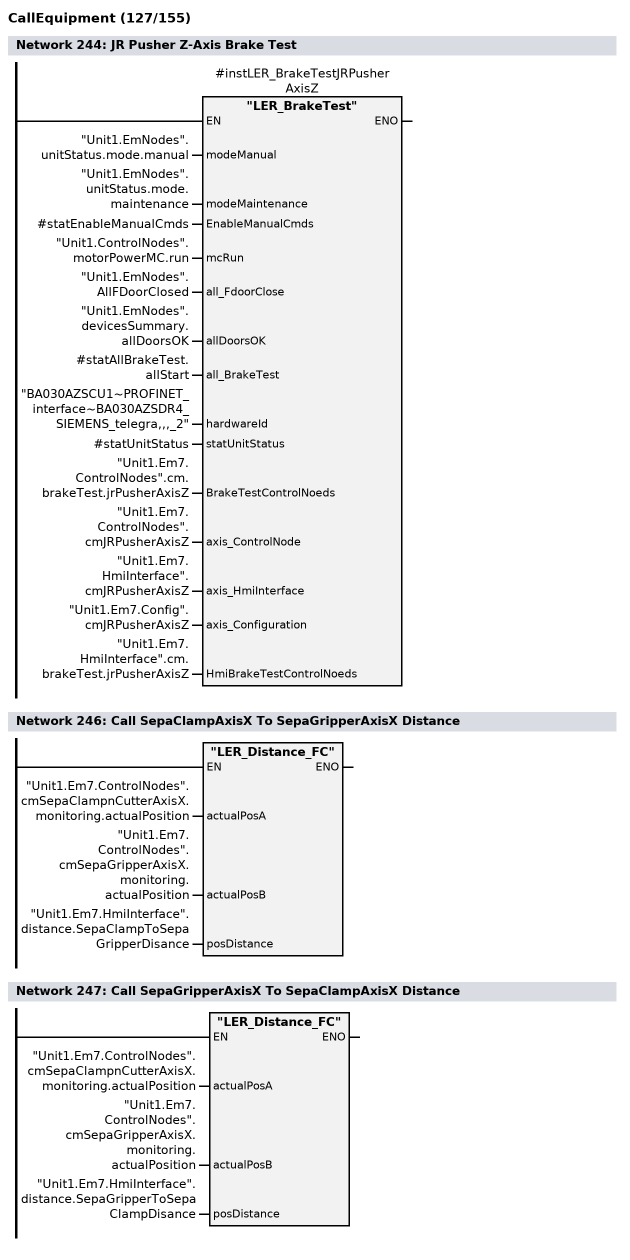
   RUNG wire#powerrail
      #instLER_BrakeTestJRPusherAxisZ(modeManual := "Unit1.EmNodes".unitStatus.mode.manual, modeMaintenance := "Unit1.EmNodes".unitStatus.mode.maintenance, EnableManualCmds := #statEnableManualCmds, mcRun := "Unit1.ControlNodes".motorPowerMC.run, all_FdoorClose := "Unit1.EmNodes".AllFDoorClosed, allDoorsOK := "Unit1.EmNodes".devicesSummary.allDoorsOK, all_BrakeTest := #statAllBrakeTest.allStart, hardwareId := "BA030AZSCU1~PROFINET_interface~BA030AZSDR4_SIEMENS_telegra,,,_2", statUnitStatus := #statUnitStatus, BrakeTestControlNoeds := "Unit1.Em7.ControlNodes".cm.brakeTest.jrPusherAxisZ, axis_ControlNode := "Unit1.Em7.ControlNodes".cmJRPusherAxisZ, axis_HmiInterface := "Unit1.Em7.HmiInterface".cmJRPusherAxisZ, axis_Configuration := "Unit1.Em7.Config".cmJRPusherAxisZ, HmiBrakeTestControlNoeds := "Unit1.Em7.HmiInterface".cm.brakeTest.jrPusherAxisZ)
   END_RUNG
   // the same network as SCL:
   #instLER_BrakeTestJRPusherAxisZ(modeManual := "Unit1.EmNodes".unitStatus.mode.manual,   // "LER_BrakeTest"
                           modeMaintenance := "Unit1.EmNodes".unitStatus.mode.maintenance,
                           EnableManualCmds := #statEnableManualCmds,
                           mcRun := "Unit1.ControlNodes".motorPowerMC.run,
                           all_FdoorClose := "Unit1.EmNodes".AllFDoorClosed,
                           allDoorsOK := "Unit1.EmNodes".devicesSummary.allDoorsOK,
                           all_BrakeTest := #statAllBrakeTest.allStart,
                           hardwareId := "BA030AZSCU1~PROFINET_interface~BA030AZSDR4_SIEMENS_telegra,,,_2",
                           statUnitStatus := #statUnitStatus,
                           BrakeTestControlNoeds := "Unit1.Em7.ControlNodes".cm.brakeTest.jrPusherAxisZ,
                           axis_ControlNode := "Unit1.Em7.ControlNodes".cmJRPusherAxisZ,
                           axis_HmiInterface := "Unit1.Em7.HmiInterface".cmJRPusherAxisZ,
                           axis_Configuration := "Unit1.Em7.Config".cmJRPusherAxisZ,
                           HmiBrakeTestControlNoeds := "Unit1.Em7.HmiInterface".cm.brakeTest.jrPusherAxisZ);
END_REGION

REGION Network 245: ******************** Axis Distance ********************
END_REGION

REGION Network 246: Call SepaClampAxisX To SepaGripperAxisX Distance
   RUNG wire#powerrail
      "LER_Distance_FC"(actualPosA := "Unit1.Em7.ControlNodes".cmSepaClampnCutterAxisX.monitoring.actualPosition, actualPosB := "Unit1.Em7.ControlNodes".cmSepaGripperAxisX.monitoring.actualPosition, posDistance := "Unit1.Em7.HmiInterface".distance.SepaClampToSepaGripperDisance)
   END_RUNG
   // the same network as SCL:
   "LER_Distance_FC"(actualPosA := "Unit1.Em7.ControlNodes".cmSepaClampnCutterAxisX.monitoring.actualPosition,
                     actualPosB := "Unit1.Em7.ControlNodes".cmSepaGripperAxisX.monitoring.actualPosition,
                     posDistance := "Unit1.Em7.HmiInterface".distance.SepaClampToSepaGripperDisance);
END_REGION

REGION Network 247: Call SepaGripperAxisX To SepaClampAxisX Distance
   RUNG wire#powerrail
      "LER_Distance_FC"(actualPosA := "Unit1.Em7.ControlNodes".cmSepaClampnCutterAxisX.monitoring.actualPosition, actualPosB := "Unit1.Em7.ControlNodes".cmSepaGripperAxisX.monitoring.actualPosition, posDistance := "Unit1.Em7.HmiInterface".distance.SepaGripperToSepaClampDisance)
   END_RUNG
   // the same network as SCL:
   "LER_Distance_FC"(actualPosA := "Unit1.Em7.ControlNodes".cmSepaClampnCutterAxisX.monitoring.actualPosition,
                     actualPosB := "Unit1.Em7.ControlNodes".cmSepaGripperAxisX.monitoring.actualPosition,
                     posDistance := "Unit1.Em7.HmiInterface".distance.SepaGripperToSepaClampDisance);
END_REGION

REGION Network 248: ********** Control Modules (TwoWayActuator) **********
END_REGION

REGION Network 249: Reset CMS
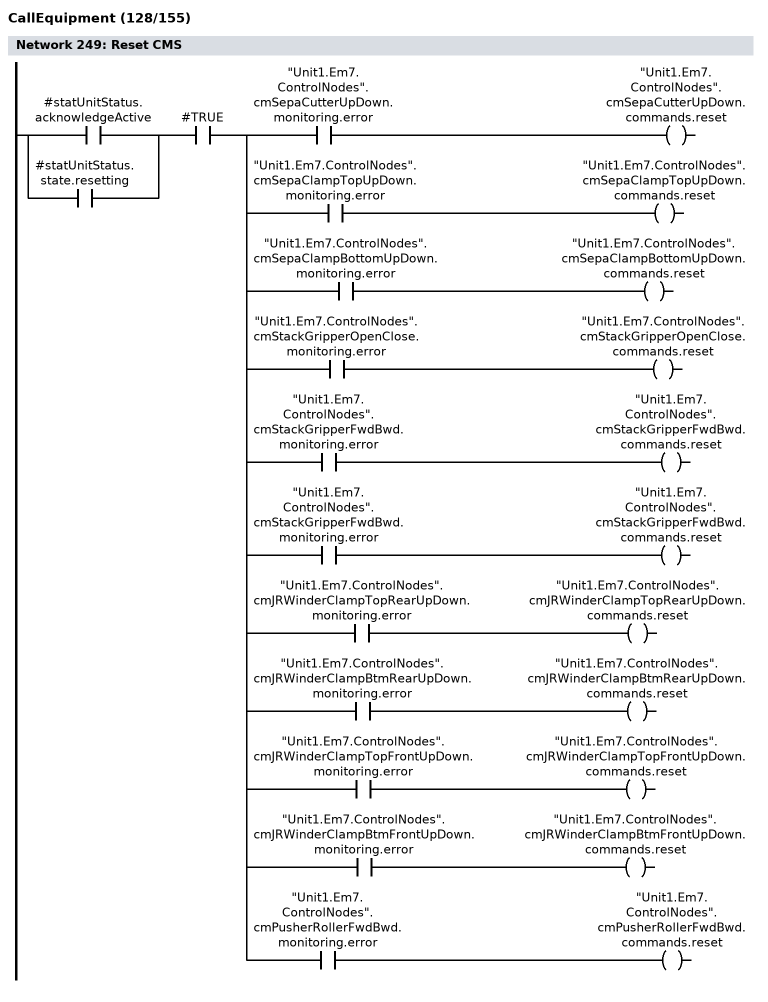
   RUNG wire#powerrail
      Contact( #statUnitStatus.acknowledgeActive )
      wire#w1
      Contact( #TRUE )
      wire#w2
      Contact( "Unit1.Em7.ControlNodes".cmSepaCutterUpDown.monitoring.error )
      Coil( "Unit1.Em7.ControlNodes".cmSepaCutterUpDown.commands.reset )
   END_RUNG
   RUNG wire#powerrail
      Contact( #statUnitStatus.state.resetting )
   END_RUNG wire#w1
   RUNG wire#w2
      Contact( "Unit1.Em7.ControlNodes".cmSepaClampTopUpDown.monitoring.error )
      Coil( "Unit1.Em7.ControlNodes".cmSepaClampTopUpDown.commands.reset )
   END_RUNG
   RUNG wire#w2
      Contact( "Unit1.Em7.ControlNodes".cmSepaClampBottomUpDown.monitoring.error )
      Coil( "Unit1.Em7.ControlNodes".cmSepaClampBottomUpDown.commands.reset )
   END_RUNG
   RUNG wire#w2
      Contact( "Unit1.Em7.ControlNodes".cmStackGripperOpenClose.monitoring.error )
      Coil( "Unit1.Em7.ControlNodes".cmStackGripperOpenClose.commands.reset )
   END_RUNG
   RUNG wire#w2
      Contact( "Unit1.Em7.ControlNodes".cmStackGripperFwdBwd.monitoring.error )
      Coil( "Unit1.Em7.ControlNodes".cmStackGripperFwdBwd.commands.reset )
   END_RUNG
   RUNG wire#w2
      Contact( "Unit1.Em7.ControlNodes".cmStackGripperFwdBwd.monitoring.error )
      Coil( "Unit1.Em7.ControlNodes".cmStackGripperFwdBwd.commands.reset )
   END_RUNG
   RUNG wire#w2
      Contact( "Unit1.Em7.ControlNodes".cmJRWinderClampTopRearUpDown.monitoring.error )
      Coil( "Unit1.Em7.ControlNodes".cmJRWinderClampTopRearUpDown.commands.reset )
   END_RUNG
   RUNG wire#w2
      Contact( "Unit1.Em7.ControlNodes".cmJRWinderClampBtmRearUpDown.monitoring.error )
      Coil( "Unit1.Em7.ControlNodes".cmJRWinderClampBtmRearUpDown.commands.reset )
   END_RUNG
   RUNG wire#w2
      Contact( "Unit1.Em7.ControlNodes".cmJRWinderClampTopFrontUpDown.monitoring.error )
      Coil( "Unit1.Em7.ControlNodes".cmJRWinderClampTopFrontUpDown.commands.reset )
   END_RUNG
   RUNG wire#w2
      Contact( "Unit1.Em7.ControlNodes".cmJRWinderClampBtmFrontUpDown.monitoring.error )
      Coil( "Unit1.Em7.ControlNodes".cmJRWinderClampBtmFrontUpDown.commands.reset )
   END_RUNG
   RUNG wire#w2
      Contact( "Unit1.Em7.ControlNodes".cmPusherRollerFwdBwd.monitoring.error )
      Coil( "Unit1.Em7.ControlNodes".cmPusherRollerFwdBwd.commands.reset )
   END_RUNG
   // the same network as SCL:
   #_w1 := (#statUnitStatus.acknowledgeActive OR #statUnitStatus.state.resetting) AND #TRUE;
   "Unit1.Em7.ControlNodes".cmSepaCutterUpDown.commands.reset := #_w1 AND "Unit1.Em7.ControlNodes".cmSepaCutterUpDown.monitoring.error;
   "Unit1.Em7.ControlNodes".cmSepaClampTopUpDown.commands.reset := #_w1 AND "Unit1.Em7.ControlNodes".cmSepaClampTopUpDown.monitoring.error;
   "Unit1.Em7.ControlNodes".cmSepaClampBottomUpDown.commands.reset := #_w1 AND "Unit1.Em7.ControlNodes".cmSepaClampBottomUpDown.monitoring.error;
   "Unit1.Em7.ControlNodes".cmStackGripperOpenClose.commands.reset := #_w1 AND "Unit1.Em7.ControlNodes".cmStackGripperOpenClose.monitoring.error;
   "Unit1.Em7.ControlNodes".cmStackGripperFwdBwd.commands.reset := #_w1 AND "Unit1.Em7.ControlNodes".cmStackGripperFwdBwd.monitoring.error;
   "Unit1.Em7.ControlNodes".cmStackGripperFwdBwd.commands.reset := #_w1 AND "Unit1.Em7.ControlNodes".cmStackGripperFwdBwd.monitoring.error;
   "Unit1.Em7.ControlNodes".cmJRWinderClampTopRearUpDown.commands.reset := #_w1 AND "Unit1.Em7.ControlNodes".cmJRWinderClampTopRearUpDown.monitoring.error;
   "Unit1.Em7.ControlNodes".cmJRWinderClampBtmRearUpDown.commands.reset := #_w1 AND "Unit1.Em7.ControlNodes".cmJRWinderClampBtmRearUpDown.monitoring.error;
   "Unit1.Em7.ControlNodes".cmJRWinderClampTopFrontUpDown.commands.reset := #_w1 AND "Unit1.Em7.ControlNodes".cmJRWinderClampTopFrontUpDown.monitoring.error;
   "Unit1.Em7.ControlNodes".cmJRWinderClampBtmFrontUpDown.commands.reset := #_w1 AND "Unit1.Em7.ControlNodes".cmJRWinderClampBtmFrontUpDown.monitoring.error;
   "Unit1.Em7.ControlNodes".cmPusherRollerFwdBwd.commands.reset := #_w1 AND "Unit1.Em7.ControlNodes".cmPusherRollerFwdBwd.monitoring.error;
END_REGION

REGION Network 251: CmSepaCutter Up
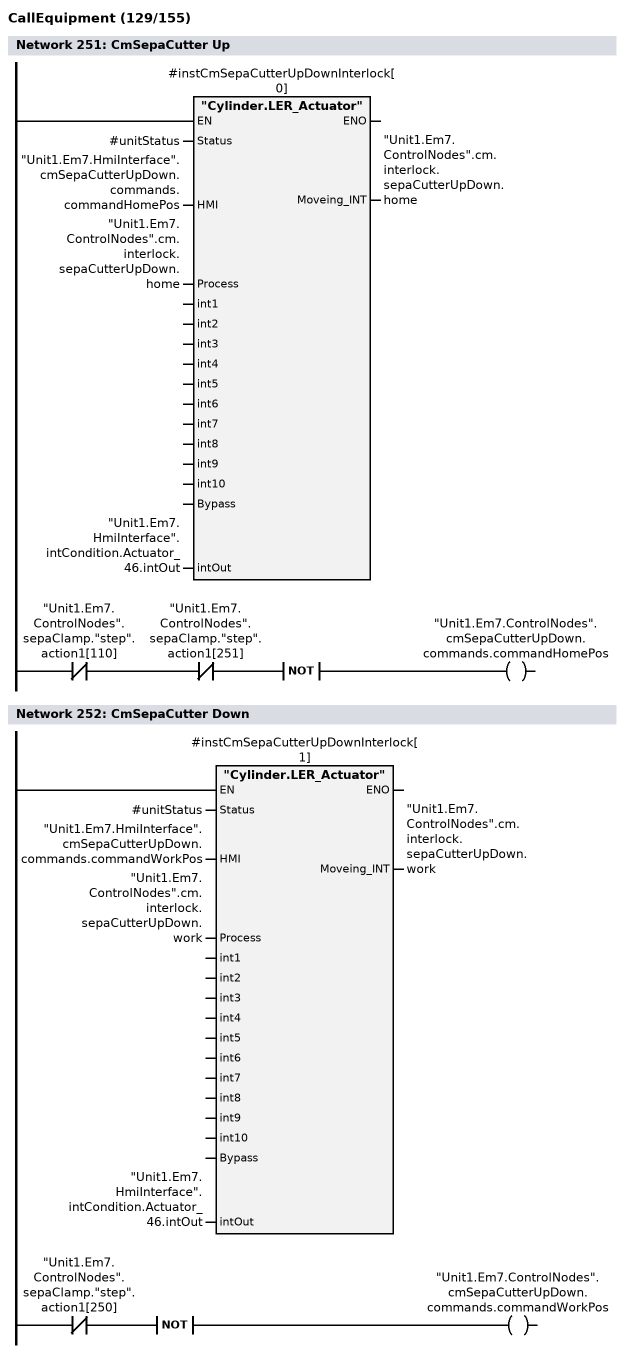
   RUNG wire#powerrail
      #instCmSepaCutterUpDownInterlock[0](Status := #unitStatus, HMI := "Unit1.Em7.HmiInterface".cmSepaCutterUpDown.commands.commandHomePos, Process := "Unit1.Em7.ControlNodes".cm.interlock.sepaCutterUpDown.home, int1 :=, int2 :=, int3 :=, int4 :=, int5 :=, int6 :=, int7 :=, int8 :=, int9 :=, int10 :=, Bypass :=, intOut := "Unit1.Em7.HmiInterface".intCondition.Actuator_46.intOut, Moveing_INT => "Unit1.Em7.ControlNodes".cm.interlock.sepaCutterUpDown.home)
   END_RUNG
   RUNG wire#powerrail
      I_Contact( "Unit1.Em7.ControlNodes".sepaClamp."step".action1[110] )
      I_Contact( "Unit1.Em7.ControlNodes".sepaClamp."step".action1[251] )
      Not()
      Coil( "Unit1.Em7.ControlNodes".cmSepaCutterUpDown.commands.commandHomePos )
   END_RUNG
   // the same network as SCL:
   #instCmSepaCutterUpDownInterlock[0](Status := #unitStatus,   // "Cylinder.LER_Actuator"
                           HMI := "Unit1.Em7.HmiInterface".cmSepaCutterUpDown.commands.commandHomePos,
                           Process := "Unit1.Em7.ControlNodes".cm.interlock.sepaCutterUpDown.home,
                           intOut := "Unit1.Em7.HmiInterface".intCondition.Actuator_46.intOut,
                           Moveing_INT => "Unit1.Em7.ControlNodes".cm.interlock.sepaCutterUpDown.home);
   "Unit1.Em7.ControlNodes".cmSepaCutterUpDown.commands.commandHomePos := NOT (NOT "Unit1.Em7.ControlNodes".sepaClamp."step".action1[110] AND NOT "Unit1.Em7.ControlNodes".sepaClamp."step".action1[251]);
END_REGION

REGION Network 252: CmSepaCutter Down
   RUNG wire#powerrail
      #instCmSepaCutterUpDownInterlock[1](Status := #unitStatus, HMI := "Unit1.Em7.HmiInterface".cmSepaCutterUpDown.commands.commandWorkPos, Process := "Unit1.Em7.ControlNodes".cm.interlock.sepaCutterUpDown.work, int1 :=, int2 :=, int3 :=, int4 :=, int5 :=, int6 :=, int7 :=, int8 :=, int9 :=, int10 :=, Bypass :=, intOut := "Unit1.Em7.HmiInterface".intCondition.Actuator_46.intOut, Moveing_INT => "Unit1.Em7.ControlNodes".cm.interlock.sepaCutterUpDown.work)
   END_RUNG
   RUNG wire#powerrail
      I_Contact( "Unit1.Em7.ControlNodes".sepaClamp."step".action1[250] )
      Not()
      Coil( "Unit1.Em7.ControlNodes".cmSepaCutterUpDown.commands.commandWorkPos )
   END_RUNG
   // the same network as SCL:
   #instCmSepaCutterUpDownInterlock[1](Status := #unitStatus,   // "Cylinder.LER_Actuator"
                           HMI := "Unit1.Em7.HmiInterface".cmSepaCutterUpDown.commands.commandWorkPos,
                           Process := "Unit1.Em7.ControlNodes".cm.interlock.sepaCutterUpDown.work,
                           intOut := "Unit1.Em7.HmiInterface".intCondition.Actuator_46.intOut,
                           Moveing_INT => "Unit1.Em7.ControlNodes".cm.interlock.sepaCutterUpDown.work);
   "Unit1.Em7.ControlNodes".cmSepaCutterUpDown.commands.commandWorkPos := NOT (NOT "Unit1.Em7.ControlNodes".sepaClamp."step".action1[250]);
END_REGION

REGION Network 253: Call instCmSepaCutterUpDown (LBC_TwoWayActuator)
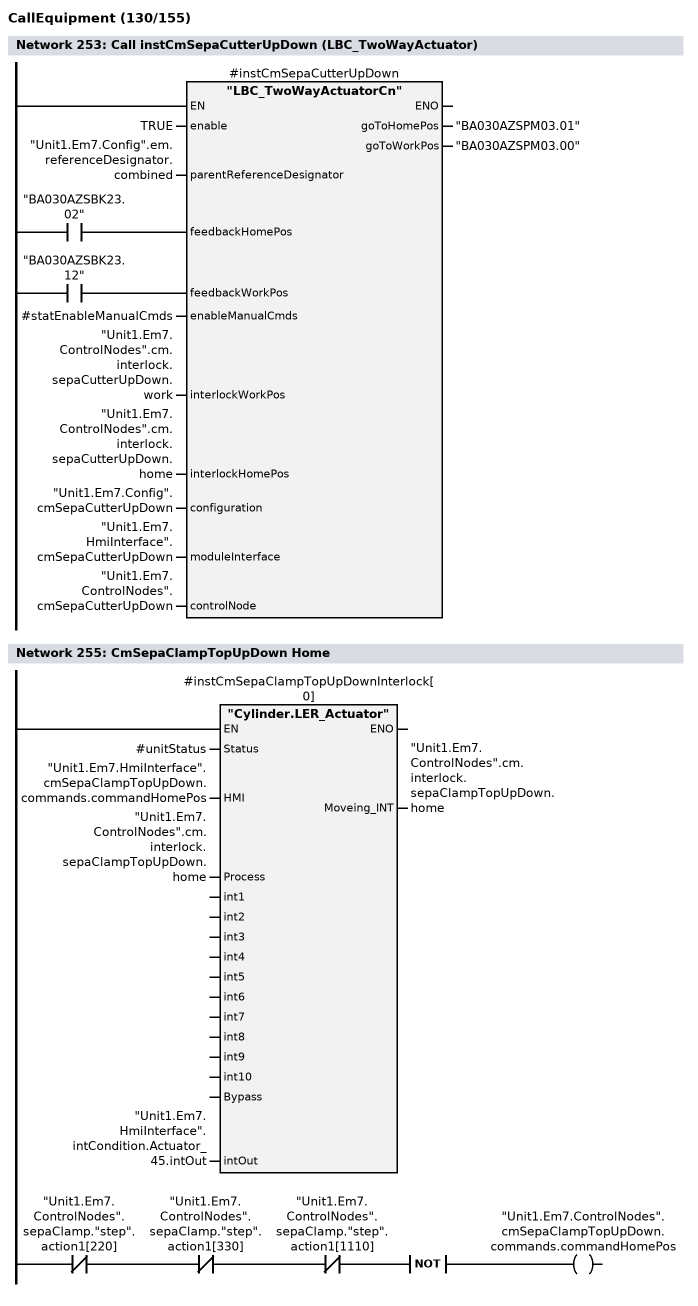
   RUNG wire#powerrail
      #instCmSepaCutterUpDown(feedbackHomePos := wire#w1, feedbackWorkPos := wire#w2, enable := TRUE, parentReferenceDesignator := "Unit1.Em7.Config".em.referenceDesignator.combined, enableManualCmds := #statEnableManualCmds, interlockWorkPos := "Unit1.Em7.ControlNodes".cm.interlock.sepaCutterUpDown.work, interlockHomePos := "Unit1.Em7.ControlNodes".cm.interlock.sepaCutterUpDown.home, configuration := "Unit1.Em7.Config".cmSepaCutterUpDown, moduleInterface := "Unit1.Em7.HmiInterface".cmSepaCutterUpDown, controlNode := "Unit1.Em7.ControlNodes".cmSepaCutterUpDown, goToHomePos => "BA030AZSPM03.01", goToWorkPos => "BA030AZSPM03.00")
   END_RUNG
   RUNG wire#powerrail
      Contact( "BA030AZSBK23.02" )
   END_RUNG wire#w1
   RUNG wire#powerrail
      Contact( "BA030AZSBK23.12" )
   END_RUNG wire#w2
   // the same network as SCL:
   #instCmSepaCutterUpDown(enable := TRUE,   // "LBC_TwoWayActuatorCn"
                           parentReferenceDesignator := "Unit1.Em7.Config".em.referenceDesignator.combined,
                           feedbackHomePos := "BA030AZSBK23.02",
                           feedbackWorkPos := "BA030AZSBK23.12",
                           enableManualCmds := #statEnableManualCmds,
                           interlockWorkPos := "Unit1.Em7.ControlNodes".cm.interlock.sepaCutterUpDown.work,
                           interlockHomePos := "Unit1.Em7.ControlNodes".cm.interlock.sepaCutterUpDown.home,
                           configuration := "Unit1.Em7.Config".cmSepaCutterUpDown,
                           moduleInterface := "Unit1.Em7.HmiInterface".cmSepaCutterUpDown,
                           controlNode := "Unit1.Em7.ControlNodes".cmSepaCutterUpDown,
                           goToHomePos => "BA030AZSPM03.01",
                           goToWorkPos => "BA030AZSPM03.00");
END_REGION

REGION Network 255: CmSepaClampTopUpDown Home
   RUNG wire#powerrail
      #instCmSepaClampTopUpDownInterlock[0](Status := #unitStatus, HMI := "Unit1.Em7.HmiInterface".cmSepaClampTopUpDown.commands.commandHomePos, Process := "Unit1.Em7.ControlNodes".cm.interlock.sepaClampTopUpDown.home, int1 :=, int2 :=, int3 :=, int4 :=, int5 :=, int6 :=, int7 :=, int8 :=, int9 :=, int10 :=, Bypass :=, intOut := "Unit1.Em7.HmiInterface".intCondition.Actuator_45.intOut, Moveing_INT => "Unit1.Em7.ControlNodes".cm.interlock.sepaClampTopUpDown.home)
   END_RUNG
   RUNG wire#powerrail
      I_Contact( "Unit1.Em7.ControlNodes".sepaClamp."step".action1[220] )
      I_Contact( "Unit1.Em7.ControlNodes".sepaClamp."step".action1[330] )
      I_Contact( "Unit1.Em7.ControlNodes".sepaClamp."step".action1[1110] )
      Not()
      Coil( "Unit1.Em7.ControlNodes".cmSepaClampTopUpDown.commands.commandHomePos )
   END_RUNG
   // the same network as SCL:
   #instCmSepaClampTopUpDownInterlock[0](Status := #unitStatus,   // "Cylinder.LER_Actuator"
                           HMI := "Unit1.Em7.HmiInterface".cmSepaClampTopUpDown.commands.commandHomePos,
                           Process := "Unit1.Em7.ControlNodes".cm.interlock.sepaClampTopUpDown.home,
                           intOut := "Unit1.Em7.HmiInterface".intCondition.Actuator_45.intOut,
                           Moveing_INT => "Unit1.Em7.ControlNodes".cm.interlock.sepaClampTopUpDown.home);
   "Unit1.Em7.ControlNodes".cmSepaClampTopUpDown.commands.commandHomePos := NOT (NOT "Unit1.Em7.ControlNodes".sepaClamp."step".action1[220] AND NOT "Unit1.Em7.ControlNodes".sepaClamp."step".action1[330] AND NOT "Unit1.Em7.ControlNodes".sepaClamp."step".action1[1110]);
END_REGION

REGION Network 256: CmSepaClampTopUpDown Work
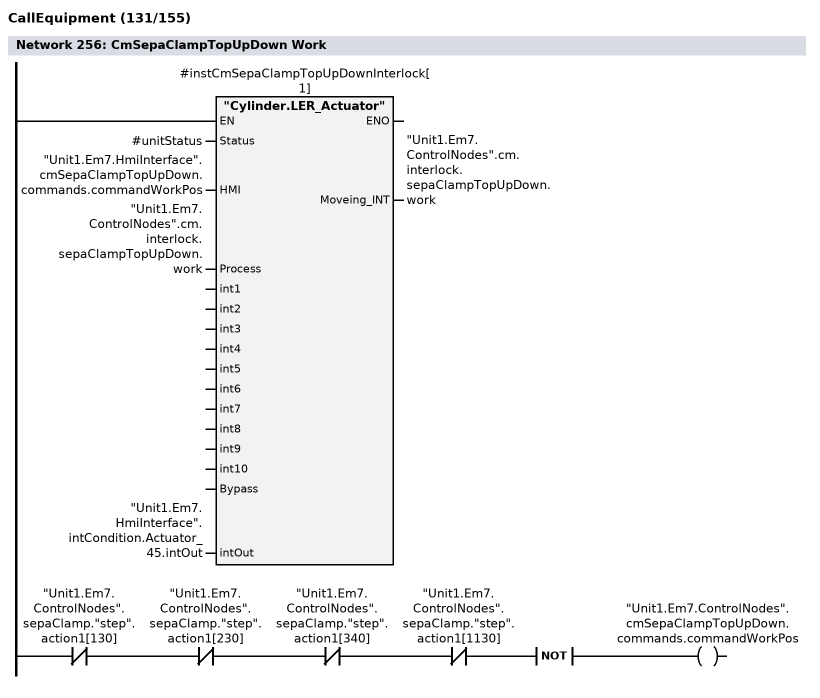
   RUNG wire#powerrail
      #instCmSepaClampTopUpDownInterlock[1](Status := #unitStatus, HMI := "Unit1.Em7.HmiInterface".cmSepaClampTopUpDown.commands.commandWorkPos, Process := "Unit1.Em7.ControlNodes".cm.interlock.sepaClampTopUpDown.work, int1 :=, int2 :=, int3 :=, int4 :=, int5 :=, int6 :=, int7 :=, int8 :=, int9 :=, int10 :=, Bypass :=, intOut := "Unit1.Em7.HmiInterface".intCondition.Actuator_45.intOut, Moveing_INT => "Unit1.Em7.ControlNodes".cm.interlock.sepaClampTopUpDown.work)
   END_RUNG
   RUNG wire#powerrail
      I_Contact( "Unit1.Em7.ControlNodes".sepaClamp."step".action1[130] )
      I_Contact( "Unit1.Em7.ControlNodes".sepaClamp."step".action1[230] )
      I_Contact( "Unit1.Em7.ControlNodes".sepaClamp."step".action1[340] )
      I_Contact( "Unit1.Em7.ControlNodes".sepaClamp."step".action1[1130] )
      Not()
      Coil( "Unit1.Em7.ControlNodes".cmSepaClampTopUpDown.commands.commandWorkPos )
   END_RUNG
   // the same network as SCL:
   #instCmSepaClampTopUpDownInterlock[1](Status := #unitStatus,   // "Cylinder.LER_Actuator"
                           HMI := "Unit1.Em7.HmiInterface".cmSepaClampTopUpDown.commands.commandWorkPos,
                           Process := "Unit1.Em7.ControlNodes".cm.interlock.sepaClampTopUpDown.work,
                           intOut := "Unit1.Em7.HmiInterface".intCondition.Actuator_45.intOut,
                           Moveing_INT => "Unit1.Em7.ControlNodes".cm.interlock.sepaClampTopUpDown.work);
   "Unit1.Em7.ControlNodes".cmSepaClampTopUpDown.commands.commandWorkPos := NOT (NOT "Unit1.Em7.ControlNodes".sepaClamp."step".action1[130] AND NOT "Unit1.Em7.ControlNodes".sepaClamp."step".action1[230] AND NOT "Unit1.Em7.ControlNodes".sepaClamp."step".action1[340] AND NOT "Unit1.Em7.ControlNodes".sepaClamp."step".action1[1130]);
END_REGION

REGION Network 257: Call instCmSepaClampTopUpDown (LBC_TwoWayActuator)
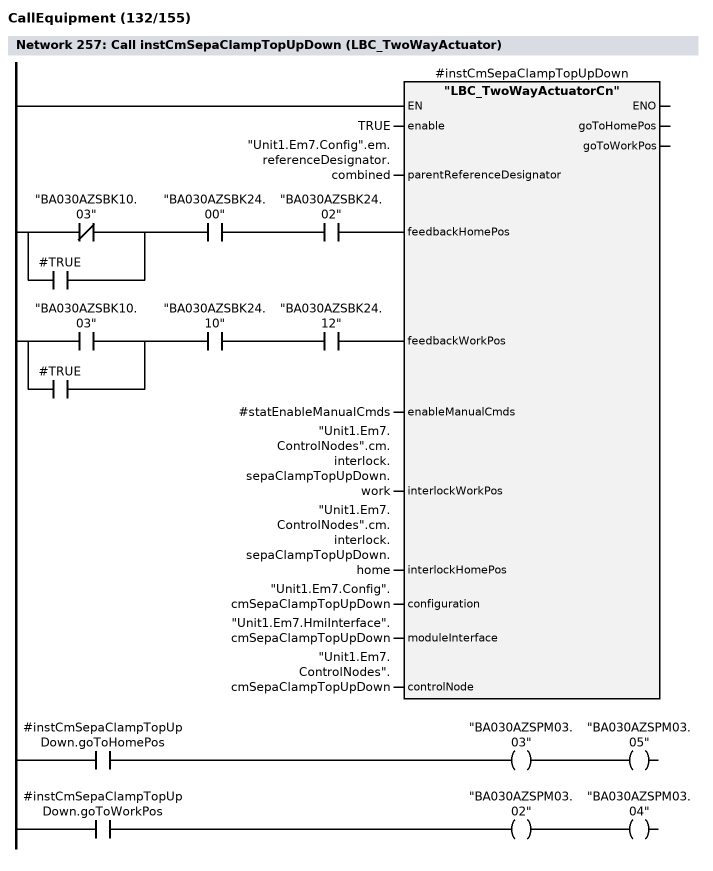
   RUNG wire#powerrail
      #instCmSepaClampTopUpDown(feedbackHomePos := wire#w2, feedbackWorkPos := wire#w4, enable := TRUE, parentReferenceDesignator := "Unit1.Em7.Config".em.referenceDesignator.combined, enableManualCmds := #statEnableManualCmds, interlockWorkPos := "Unit1.Em7.ControlNodes".cm.interlock.sepaClampTopUpDown.work, interlockHomePos := "Unit1.Em7.ControlNodes".cm.interlock.sepaClampTopUpDown.home, configuration := "Unit1.Em7.Config".cmSepaClampTopUpDown, moduleInterface := "Unit1.Em7.HmiInterface".cmSepaClampTopUpDown, controlNode := "Unit1.Em7.ControlNodes".cmSepaClampTopUpDown, goToHomePos =>, goToWorkPos =>)
   END_RUNG
   RUNG wire#powerrail
      I_Contact( "BA030AZSBK10.03" )
      wire#w1
      Contact( "BA030AZSBK24.00" )
      Contact( "BA030AZSBK24.02" )
   END_RUNG wire#w2
   RUNG wire#powerrail
      Contact( #TRUE )
   END_RUNG wire#w1
   RUNG wire#powerrail
      Contact( "BA030AZSBK10.03" )
      wire#w3
      Contact( "BA030AZSBK24.10" )
      Contact( "BA030AZSBK24.12" )
   END_RUNG wire#w4
   RUNG wire#powerrail
      Contact( #TRUE )
   END_RUNG wire#w3
   RUNG wire#powerrail
      Contact( #instCmSepaClampTopUpDown.goToHomePos )
      Coil( "BA030AZSPM03.03" )
      Coil( "BA030AZSPM03.05" )
   END_RUNG
   RUNG wire#powerrail
      Contact( #instCmSepaClampTopUpDown.goToWorkPos )
      Coil( "BA030AZSPM03.02" )
      Coil( "BA030AZSPM03.04" )
   END_RUNG
   // the same network as SCL:
   #instCmSepaClampTopUpDown(enable := TRUE,   // "LBC_TwoWayActuatorCn"
                           parentReferenceDesignator := "Unit1.Em7.Config".em.referenceDesignator.combined,
                           feedbackHomePos := (NOT "BA030AZSBK10.03" OR #TRUE) AND "BA030AZSBK24.00" AND "BA030AZSBK24.02",
                           feedbackWorkPos := ("BA030AZSBK10.03" OR #TRUE) AND "BA030AZSBK24.10" AND "BA030AZSBK24.12",
                           enableManualCmds := #statEnableManualCmds,
                           interlockWorkPos := "Unit1.Em7.ControlNodes".cm.interlock.sepaClampTopUpDown.work,
                           interlockHomePos := "Unit1.Em7.ControlNodes".cm.interlock.sepaClampTopUpDown.home,
                           configuration := "Unit1.Em7.Config".cmSepaClampTopUpDown,
                           moduleInterface := "Unit1.Em7.HmiInterface".cmSepaClampTopUpDown,
                           controlNode := "Unit1.Em7.ControlNodes".cmSepaClampTopUpDown);
   "BA030AZSPM03.03" := #instCmSepaClampTopUpDown.goToHomePos;
   "BA030AZSPM03.05" := #instCmSepaClampTopUpDown.goToHomePos;
   "BA030AZSPM03.02" := #instCmSepaClampTopUpDown.goToWorkPos;
   "BA030AZSPM03.04" := #instCmSepaClampTopUpDown.goToWorkPos;
END_REGION

REGION Network 259: CmSepaClampBottomUpDown Home
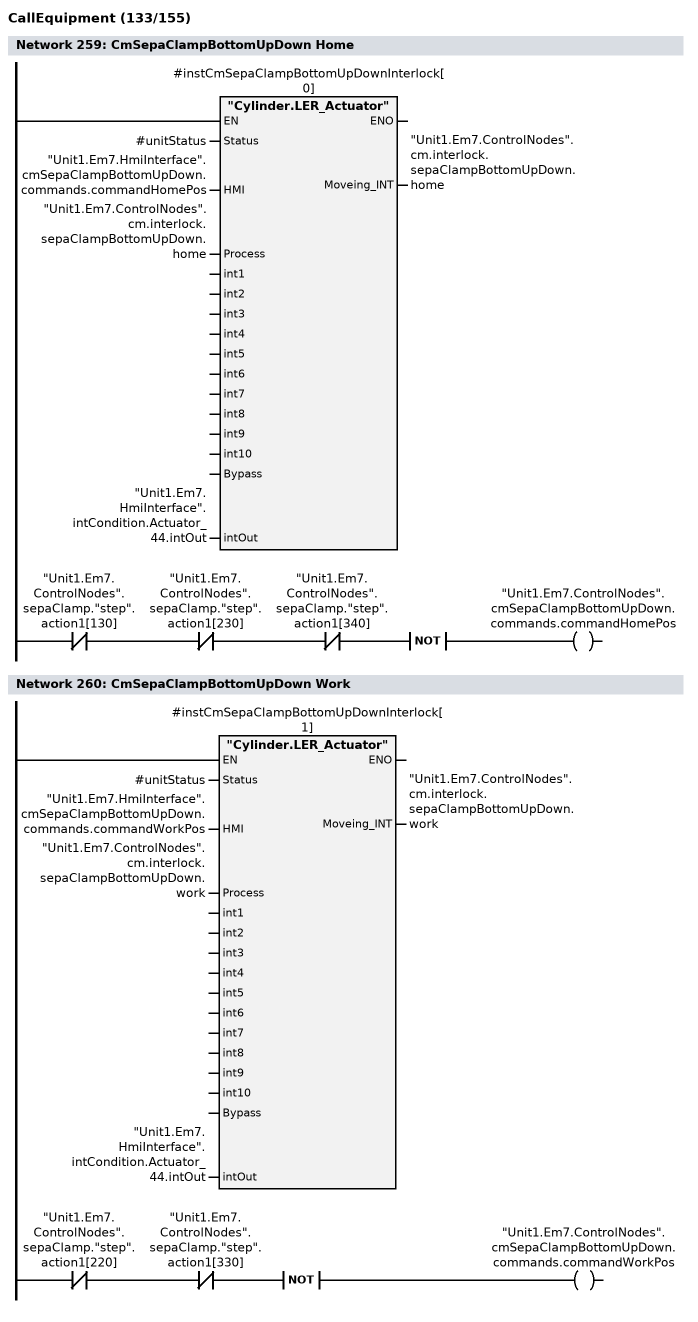
   RUNG wire#powerrail
      #instCmSepaClampBottomUpDownInterlock[0](Status := #unitStatus, HMI := "Unit1.Em7.HmiInterface".cmSepaClampBottomUpDown.commands.commandHomePos, Process := "Unit1.Em7.ControlNodes".cm.interlock.sepaClampBottomUpDown.home, int1 :=, int2 :=, int3 :=, int4 :=, int5 :=, int6 :=, int7 :=, int8 :=, int9 :=, int10 :=, Bypass :=, intOut := "Unit1.Em7.HmiInterface".intCondition.Actuator_44.intOut, Moveing_INT => "Unit1.Em7.ControlNodes".cm.interlock.sepaClampBottomUpDown.home)
   END_RUNG
   RUNG wire#powerrail
      I_Contact( "Unit1.Em7.ControlNodes".sepaClamp."step".action1[130] )
      I_Contact( "Unit1.Em7.ControlNodes".sepaClamp."step".action1[230] )
      I_Contact( "Unit1.Em7.ControlNodes".sepaClamp."step".action1[340] )
      Not()
      Coil( "Unit1.Em7.ControlNodes".cmSepaClampBottomUpDown.commands.commandHomePos )
   END_RUNG
   // the same network as SCL:
   #instCmSepaClampBottomUpDownInterlock[0](Status := #unitStatus,   // "Cylinder.LER_Actuator"
                           HMI := "Unit1.Em7.HmiInterface".cmSepaClampBottomUpDown.commands.commandHomePos,
                           Process := "Unit1.Em7.ControlNodes".cm.interlock.sepaClampBottomUpDown.home,
                           intOut := "Unit1.Em7.HmiInterface".intCondition.Actuator_44.intOut,
                           Moveing_INT => "Unit1.Em7.ControlNodes".cm.interlock.sepaClampBottomUpDown.home);
   "Unit1.Em7.ControlNodes".cmSepaClampBottomUpDown.commands.commandHomePos := NOT (NOT "Unit1.Em7.ControlNodes".sepaClamp."step".action1[130] AND NOT "Unit1.Em7.ControlNodes".sepaClamp."step".action1[230] AND NOT "Unit1.Em7.ControlNodes".sepaClamp."step".action1[340]);
END_REGION

REGION Network 260: CmSepaClampBottomUpDown Work
   RUNG wire#powerrail
      #instCmSepaClampBottomUpDownInterlock[1](Status := #unitStatus, HMI := "Unit1.Em7.HmiInterface".cmSepaClampBottomUpDown.commands.commandWorkPos, Process := "Unit1.Em7.ControlNodes".cm.interlock.sepaClampBottomUpDown.work, int1 :=, int2 :=, int3 :=, int4 :=, int5 :=, int6 :=, int7 :=, int8 :=, int9 :=, int10 :=, Bypass :=, intOut := "Unit1.Em7.HmiInterface".intCondition.Actuator_44.intOut, Moveing_INT => "Unit1.Em7.ControlNodes".cm.interlock.sepaClampBottomUpDown.work)
   END_RUNG
   RUNG wire#powerrail
      I_Contact( "Unit1.Em7.ControlNodes".sepaClamp."step".action1[220] )
      I_Contact( "Unit1.Em7.ControlNodes".sepaClamp."step".action1[330] )
      Not()
      Coil( "Unit1.Em7.ControlNodes".cmSepaClampBottomUpDown.commands.commandWorkPos )
   END_RUNG
   // the same network as SCL:
   #instCmSepaClampBottomUpDownInterlock[1](Status := #unitStatus,   // "Cylinder.LER_Actuator"
                           HMI := "Unit1.Em7.HmiInterface".cmSepaClampBottomUpDown.commands.commandWorkPos,
                           Process := "Unit1.Em7.ControlNodes".cm.interlock.sepaClampBottomUpDown.work,
                           intOut := "Unit1.Em7.HmiInterface".intCondition.Actuator_44.intOut,
                           Moveing_INT => "Unit1.Em7.ControlNodes".cm.interlock.sepaClampBottomUpDown.work);
   "Unit1.Em7.ControlNodes".cmSepaClampBottomUpDown.commands.commandWorkPos := NOT (NOT "Unit1.Em7.ControlNodes".sepaClamp."step".action1[220] AND NOT "Unit1.Em7.ControlNodes".sepaClamp."step".action1[330]);
END_REGION

REGION Network 261: Call instCmSepaClampBottomUpDown (LBC_TwoWayActuator)
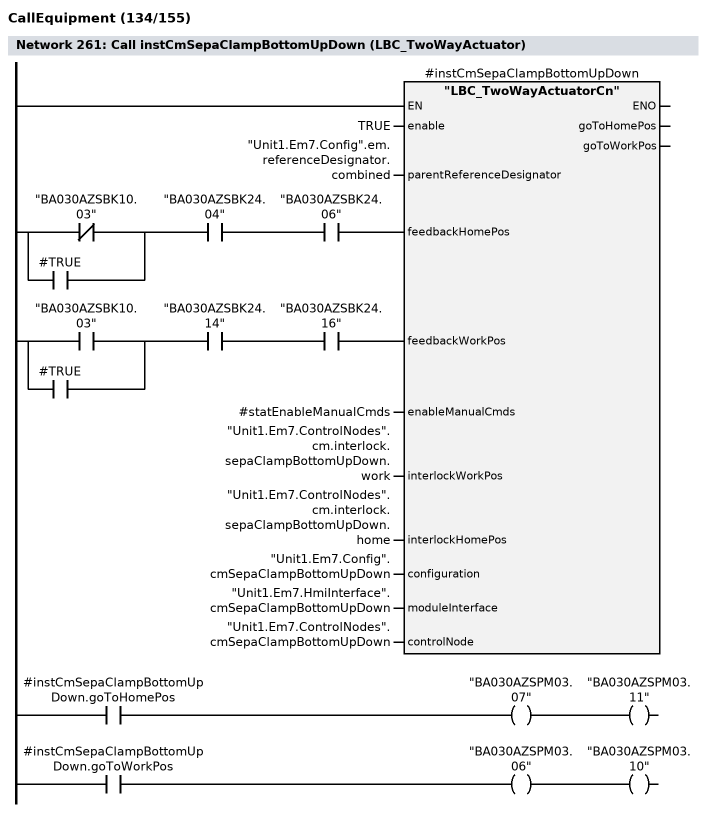
   RUNG wire#powerrail
      #instCmSepaClampBottomUpDown(feedbackHomePos := wire#w2, feedbackWorkPos := wire#w4, enable := TRUE, parentReferenceDesignator := "Unit1.Em7.Config".em.referenceDesignator.combined, enableManualCmds := #statEnableManualCmds, interlockWorkPos := "Unit1.Em7.ControlNodes".cm.interlock.sepaClampBottomUpDown.work, interlockHomePos := "Unit1.Em7.ControlNodes".cm.interlock.sepaClampBottomUpDown.home, configuration := "Unit1.Em7.Config".cmSepaClampBottomUpDown, moduleInterface := "Unit1.Em7.HmiInterface".cmSepaClampBottomUpDown, controlNode := "Unit1.Em7.ControlNodes".cmSepaClampBottomUpDown, goToHomePos =>, goToWorkPos =>)
   END_RUNG
   RUNG wire#powerrail
      I_Contact( "BA030AZSBK10.03" )
      wire#w1
      Contact( "BA030AZSBK24.04" )
      Contact( "BA030AZSBK24.06" )
   END_RUNG wire#w2
   RUNG wire#powerrail
      Contact( #TRUE )
   END_RUNG wire#w1
   RUNG wire#powerrail
      Contact( "BA030AZSBK10.03" )
      wire#w3
      Contact( "BA030AZSBK24.14" )
      Contact( "BA030AZSBK24.16" )
   END_RUNG wire#w4
   RUNG wire#powerrail
      Contact( #TRUE )
   END_RUNG wire#w3
   RUNG wire#powerrail
      Contact( #instCmSepaClampBottomUpDown.goToHomePos )
      Coil( "BA030AZSPM03.07" )
      Coil( "BA030AZSPM03.11" )
   END_RUNG
   RUNG wire#powerrail
      Contact( #instCmSepaClampBottomUpDown.goToWorkPos )
      Coil( "BA030AZSPM03.06" )
      Coil( "BA030AZSPM03.10" )
   END_RUNG
   // the same network as SCL:
   #instCmSepaClampBottomUpDown(enable := TRUE,   // "LBC_TwoWayActuatorCn"
                           parentReferenceDesignator := "Unit1.Em7.Config".em.referenceDesignator.combined,
                           feedbackHomePos := (NOT "BA030AZSBK10.03" OR #TRUE) AND "BA030AZSBK24.04" AND "BA030AZSBK24.06",
                           feedbackWorkPos := ("BA030AZSBK10.03" OR #TRUE) AND "BA030AZSBK24.14" AND "BA030AZSBK24.16",
                           enableManualCmds := #statEnableManualCmds,
                           interlockWorkPos := "Unit1.Em7.ControlNodes".cm.interlock.sepaClampBottomUpDown.work,
                           interlockHomePos := "Unit1.Em7.ControlNodes".cm.interlock.sepaClampBottomUpDown.home,
                           configuration := "Unit1.Em7.Config".cmSepaClampBottomUpDown,
                           moduleInterface := "Unit1.Em7.HmiInterface".cmSepaClampBottomUpDown,
                           controlNode := "Unit1.Em7.ControlNodes".cmSepaClampBottomUpDown);
   "BA030AZSPM03.07" := #instCmSepaClampBottomUpDown.goToHomePos;
   "BA030AZSPM03.11" := #instCmSepaClampBottomUpDown.goToHomePos;
   "BA030AZSPM03.06" := #instCmSepaClampBottomUpDown.goToWorkPos;
   "BA030AZSPM03.10" := #instCmSepaClampBottomUpDown.goToWorkPos;
END_REGION

REGION Network 263: StackGripperOpenClose Home
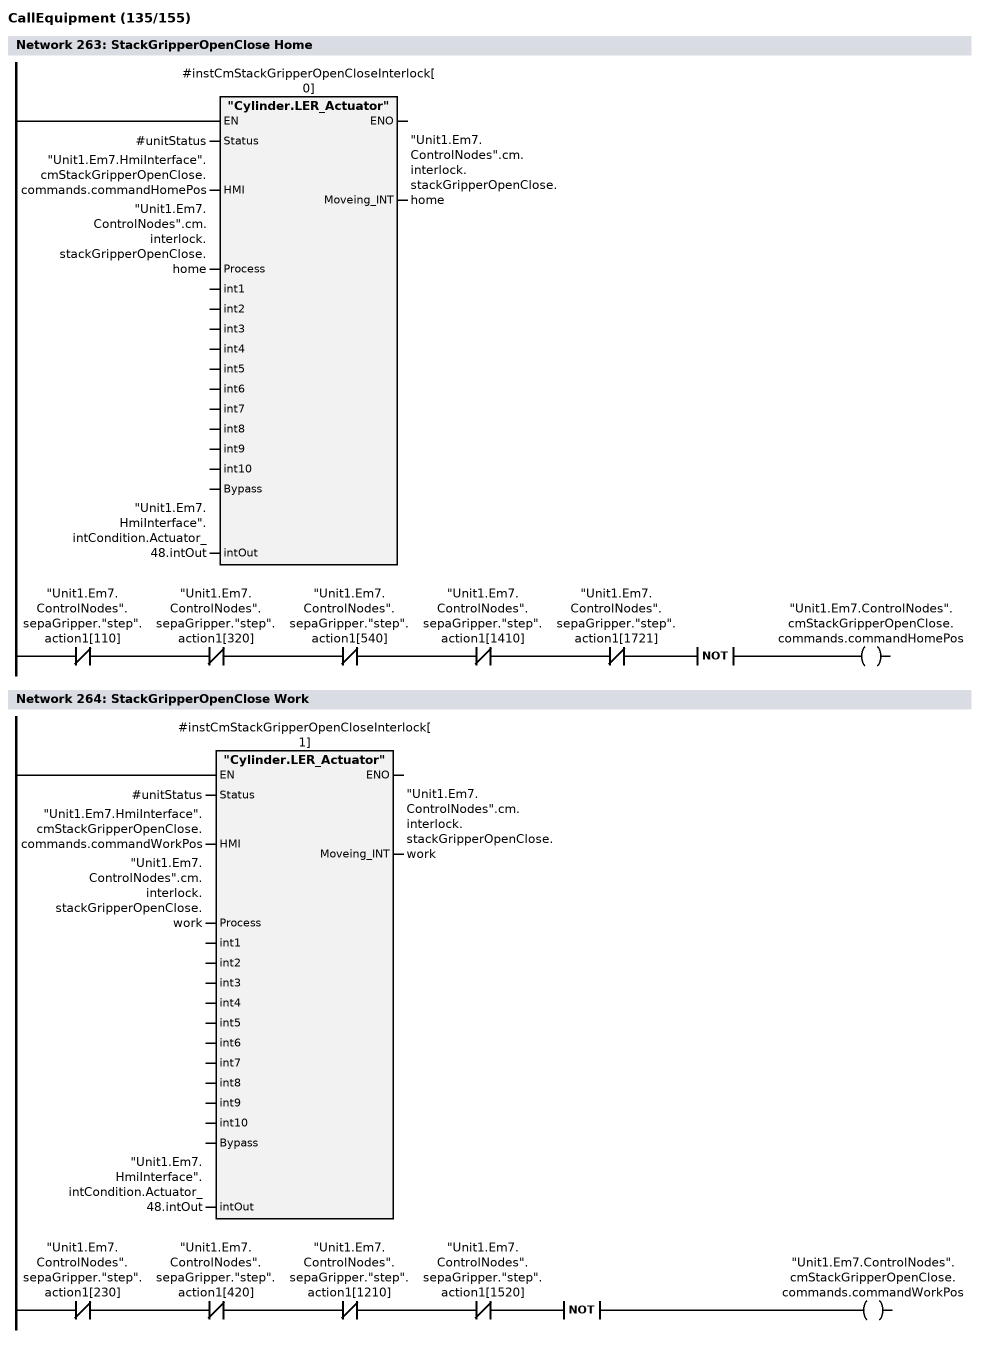
   RUNG wire#powerrail
      #instCmStackGripperOpenCloseInterlock[0](Status := #unitStatus, HMI := "Unit1.Em7.HmiInterface".cmStackGripperOpenClose.commands.commandHomePos, Process := "Unit1.Em7.ControlNodes".cm.interlock.stackGripperOpenClose.home, int1 :=, int2 :=, int3 :=, int4 :=, int5 :=, int6 :=, int7 :=, int8 :=, int9 :=, int10 :=, Bypass :=, intOut := "Unit1.Em7.HmiInterface".intCondition.Actuator_48.intOut, Moveing_INT => "Unit1.Em7.ControlNodes".cm.interlock.stackGripperOpenClose.home)
   END_RUNG
   RUNG wire#powerrail
      I_Contact( "Unit1.Em7.ControlNodes".sepaGripper."step".action1[110] )
      I_Contact( "Unit1.Em7.ControlNodes".sepaGripper."step".action1[320] )
      I_Contact( "Unit1.Em7.ControlNodes".sepaGripper."step".action1[540] )
      I_Contact( "Unit1.Em7.ControlNodes".sepaGripper."step".action1[1410] )
      I_Contact( "Unit1.Em7.ControlNodes".sepaGripper."step".action1[1721] )
      Not()
      Coil( "Unit1.Em7.ControlNodes".cmStackGripperOpenClose.commands.commandHomePos )
   END_RUNG
   // the same network as SCL:
   #instCmStackGripperOpenCloseInterlock[0](Status := #unitStatus,   // "Cylinder.LER_Actuator"
                           HMI := "Unit1.Em7.HmiInterface".cmStackGripperOpenClose.commands.commandHomePos,
                           Process := "Unit1.Em7.ControlNodes".cm.interlock.stackGripperOpenClose.home,
                           intOut := "Unit1.Em7.HmiInterface".intCondition.Actuator_48.intOut,
                           Moveing_INT => "Unit1.Em7.ControlNodes".cm.interlock.stackGripperOpenClose.home);
   "Unit1.Em7.ControlNodes".cmStackGripperOpenClose.commands.commandHomePos := NOT (NOT "Unit1.Em7.ControlNodes".sepaGripper."step".action1[110] AND NOT "Unit1.Em7.ControlNodes".sepaGripper."step".action1[320] AND NOT "Unit1.Em7.ControlNodes".sepaGripper."step".action1[540] AND NOT "Unit1.Em7.ControlNodes".sepaGripper."step".action1[1410] AND NOT "Unit1.Em7.ControlNodes".sepaGripper."step".action1[1721]);
END_REGION

REGION Network 264: StackGripperOpenClose Work
   RUNG wire#powerrail
      #instCmStackGripperOpenCloseInterlock[1](Status := #unitStatus, HMI := "Unit1.Em7.HmiInterface".cmStackGripperOpenClose.commands.commandWorkPos, Process := "Unit1.Em7.ControlNodes".cm.interlock.stackGripperOpenClose.work, int1 :=, int2 :=, int3 :=, int4 :=, int5 :=, int6 :=, int7 :=, int8 :=, int9 :=, int10 :=, Bypass :=, intOut := "Unit1.Em7.HmiInterface".intCondition.Actuator_48.intOut, Moveing_INT => "Unit1.Em7.ControlNodes".cm.interlock.stackGripperOpenClose.work)
   END_RUNG
   RUNG wire#powerrail
      I_Contact( "Unit1.Em7.ControlNodes".sepaGripper."step".action1[230] )
      I_Contact( "Unit1.Em7.ControlNodes".sepaGripper."step".action1[420] )
      I_Contact( "Unit1.Em7.ControlNodes".sepaGripper."step".action1[1210] )
      I_Contact( "Unit1.Em7.ControlNodes".sepaGripper."step".action1[1520] )
      Not()
      Coil( "Unit1.Em7.ControlNodes".cmStackGripperOpenClose.commands.commandWorkPos )
   END_RUNG
   // the same network as SCL:
   #instCmStackGripperOpenCloseInterlock[1](Status := #unitStatus,   // "Cylinder.LER_Actuator"
                           HMI := "Unit1.Em7.HmiInterface".cmStackGripperOpenClose.commands.commandWorkPos,
                           Process := "Unit1.Em7.ControlNodes".cm.interlock.stackGripperOpenClose.work,
                           intOut := "Unit1.Em7.HmiInterface".intCondition.Actuator_48.intOut,
                           Moveing_INT => "Unit1.Em7.ControlNodes".cm.interlock.stackGripperOpenClose.work);
   "Unit1.Em7.ControlNodes".cmStackGripperOpenClose.commands.commandWorkPos := NOT (NOT "Unit1.Em7.ControlNodes".sepaGripper."step".action1[230] AND NOT "Unit1.Em7.ControlNodes".sepaGripper."step".action1[420] AND NOT "Unit1.Em7.ControlNodes".sepaGripper."step".action1[1210] AND NOT "Unit1.Em7.ControlNodes".sepaGripper."step".action1[1520]);
END_REGION

REGION Network 265: Call instCmStackGripperOpenClose (LBC_TwoWayActuator)
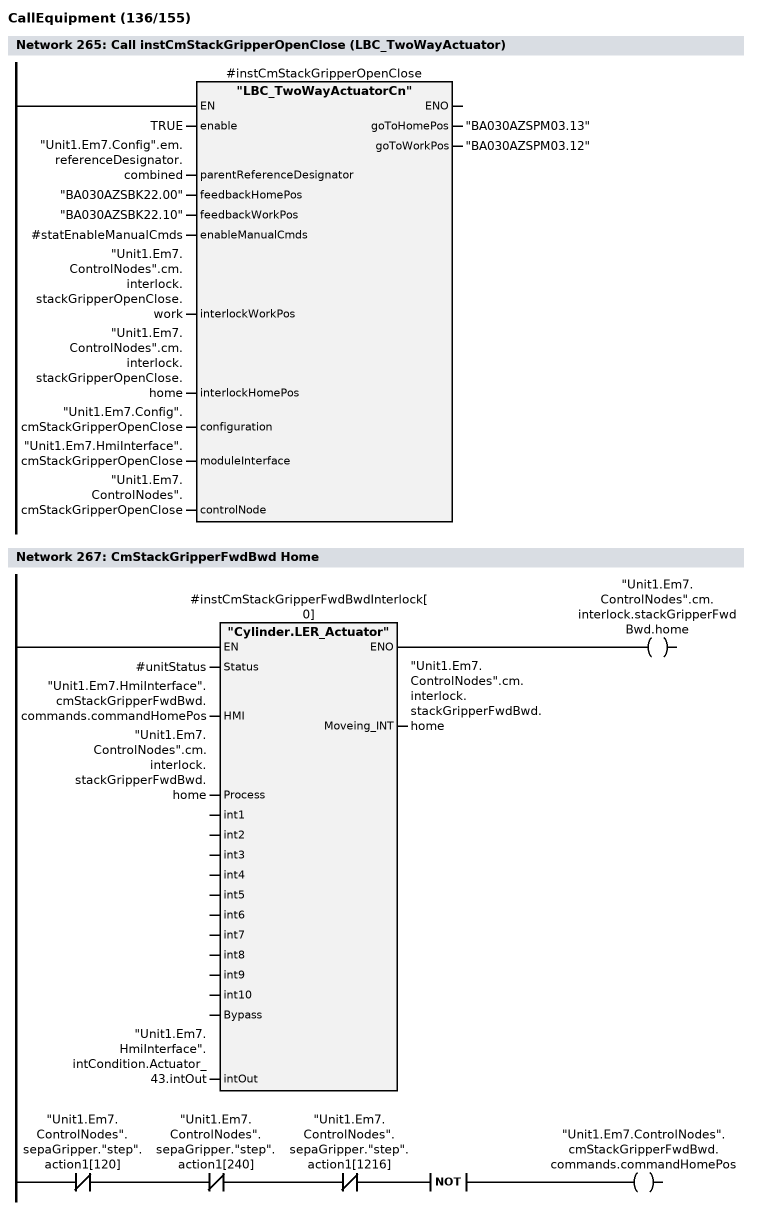
   RUNG wire#powerrail
      #instCmStackGripperOpenClose(enable := TRUE, parentReferenceDesignator := "Unit1.Em7.Config".em.referenceDesignator.combined, feedbackHomePos := "BA030AZSBK22.00", feedbackWorkPos := "BA030AZSBK22.10", enableManualCmds := #statEnableManualCmds, interlockWorkPos := "Unit1.Em7.ControlNodes".cm.interlock.stackGripperOpenClose.work, interlockHomePos := "Unit1.Em7.ControlNodes".cm.interlock.stackGripperOpenClose.home, configuration := "Unit1.Em7.Config".cmStackGripperOpenClose, moduleInterface := "Unit1.Em7.HmiInterface".cmStackGripperOpenClose, controlNode := "Unit1.Em7.ControlNodes".cmStackGripperOpenClose, goToHomePos => "BA030AZSPM03.13", goToWorkPos => "BA030AZSPM03.12")
   END_RUNG
   // the same network as SCL:
   #instCmStackGripperOpenClose(enable := TRUE,   // "LBC_TwoWayActuatorCn"
                           parentReferenceDesignator := "Unit1.Em7.Config".em.referenceDesignator.combined,
                           feedbackHomePos := "BA030AZSBK22.00",
                           feedbackWorkPos := "BA030AZSBK22.10",
                           enableManualCmds := #statEnableManualCmds,
                           interlockWorkPos := "Unit1.Em7.ControlNodes".cm.interlock.stackGripperOpenClose.work,
                           interlockHomePos := "Unit1.Em7.ControlNodes".cm.interlock.stackGripperOpenClose.home,
                           configuration := "Unit1.Em7.Config".cmStackGripperOpenClose,
                           moduleInterface := "Unit1.Em7.HmiInterface".cmStackGripperOpenClose,
                           controlNode := "Unit1.Em7.ControlNodes".cmStackGripperOpenClose,
                           goToHomePos => "BA030AZSPM03.13",
                           goToWorkPos => "BA030AZSPM03.12");
END_REGION

REGION Network 267: CmStackGripperFwdBwd Home
   RUNG wire#powerrail
      #instCmStackGripperFwdBwdInterlock[0](Status := #unitStatus, HMI := "Unit1.Em7.HmiInterface".cmStackGripperFwdBwd.commands.commandHomePos, Process := "Unit1.Em7.ControlNodes".cm.interlock.stackGripperFwdBwd.home, int1 :=, int2 :=, int3 :=, int4 :=, int5 :=, int6 :=, int7 :=, int8 :=, int9 :=, int10 :=, Bypass :=, intOut := "Unit1.Em7.HmiInterface".intCondition.Actuator_43.intOut, Moveing_INT => "Unit1.Em7.ControlNodes".cm.interlock.stackGripperFwdBwd.home)
      Coil( "Unit1.Em7.ControlNodes".cm.interlock.stackGripperFwdBwd.home )
   END_RUNG
   RUNG wire#powerrail
      I_Contact( "Unit1.Em7.ControlNodes".sepaGripper."step".action1[120] )
      I_Contact( "Unit1.Em7.ControlNodes".sepaGripper."step".action1[240] )
      I_Contact( "Unit1.Em7.ControlNodes".sepaGripper."step".action1[1216] )
      Not()
      Coil( "Unit1.Em7.ControlNodes".cmStackGripperFwdBwd.commands.commandHomePos )
   END_RUNG
   // the same network as SCL:
   #instCmStackGripperFwdBwdInterlock[0](Status := #unitStatus,   // "Cylinder.LER_Actuator"
                           HMI := "Unit1.Em7.HmiInterface".cmStackGripperFwdBwd.commands.commandHomePos,
                           Process := "Unit1.Em7.ControlNodes".cm.interlock.stackGripperFwdBwd.home,
                           intOut := "Unit1.Em7.HmiInterface".intCondition.Actuator_43.intOut,
                           Moveing_INT => "Unit1.Em7.ControlNodes".cm.interlock.stackGripperFwdBwd.home,
                           ENO => #_w1);
   "Unit1.Em7.ControlNodes".cm.interlock.stackGripperFwdBwd.home := #_w1;
   "Unit1.Em7.ControlNodes".cmStackGripperFwdBwd.commands.commandHomePos := NOT (NOT "Unit1.Em7.ControlNodes".sepaGripper."step".action1[120] AND NOT "Unit1.Em7.ControlNodes".sepaGripper."step".action1[240] AND NOT "Unit1.Em7.ControlNodes".sepaGripper."step".action1[1216]);
END_REGION

REGION Network 268: CmStackGripperFwdBwd Work
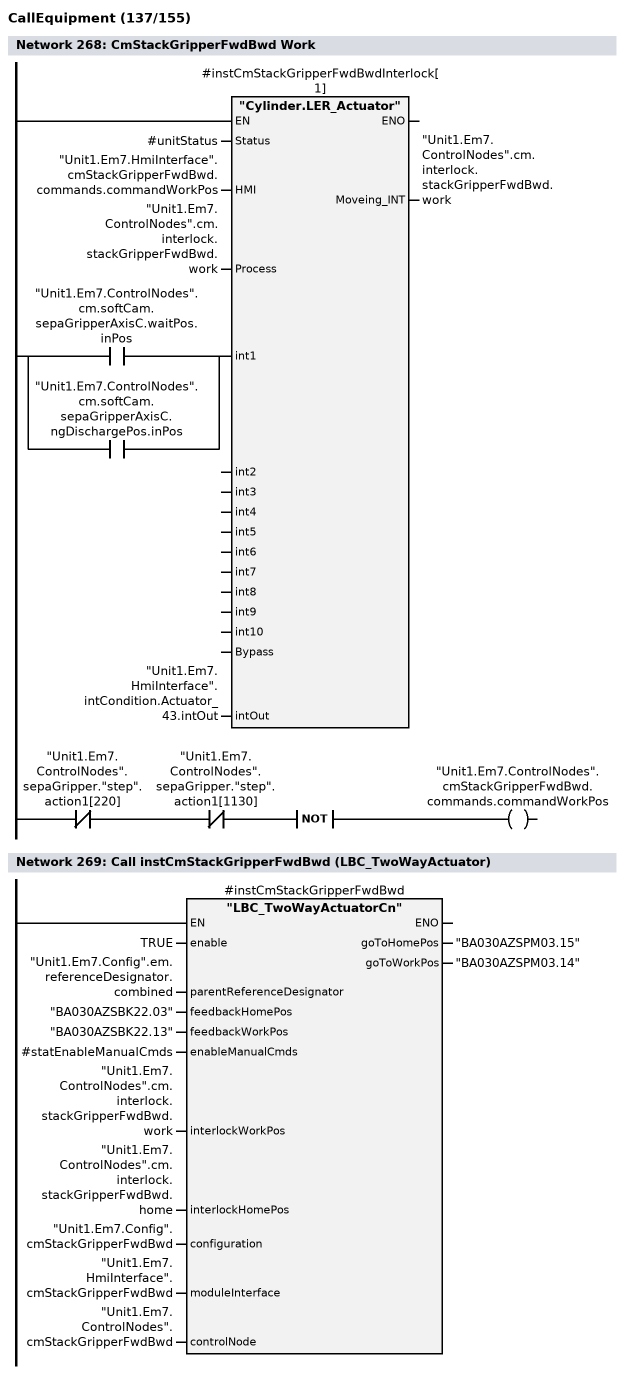
   RUNG wire#powerrail
      #instCmStackGripperFwdBwdInterlock[1](int1 := wire#w1, Status := #unitStatus, HMI := "Unit1.Em7.HmiInterface".cmStackGripperFwdBwd.commands.commandWorkPos, Process := "Unit1.Em7.ControlNodes".cm.interlock.stackGripperFwdBwd.work, int2 :=, int3 :=, int4 :=, int5 :=, int6 :=, int7 :=, int8 :=, int9 :=, int10 :=, Bypass :=, intOut := "Unit1.Em7.HmiInterface".intCondition.Actuator_43.intOut, Moveing_INT => "Unit1.Em7.ControlNodes".cm.interlock.stackGripperFwdBwd.work)
   END_RUNG
   RUNG wire#powerrail
      Contact( "Unit1.Em7.ControlNodes".cm.softCam.sepaGripperAxisC.waitPos.inPos )
   END_RUNG wire#w1
   RUNG wire#powerrail
      Contact( "Unit1.Em7.ControlNodes".cm.softCam.sepaGripperAxisC.ngDischargePos.inPos )
   END_RUNG wire#w1
   RUNG wire#powerrail
      I_Contact( "Unit1.Em7.ControlNodes".sepaGripper."step".action1[220] )
      I_Contact( "Unit1.Em7.ControlNodes".sepaGripper."step".action1[1130] )
      Not()
      Coil( "Unit1.Em7.ControlNodes".cmStackGripperFwdBwd.commands.commandWorkPos )
   END_RUNG
   // the same network as SCL:
   #instCmStackGripperFwdBwdInterlock[1](Status := #unitStatus,   // "Cylinder.LER_Actuator"
                           HMI := "Unit1.Em7.HmiInterface".cmStackGripperFwdBwd.commands.commandWorkPos,
                           Process := "Unit1.Em7.ControlNodes".cm.interlock.stackGripperFwdBwd.work,
                           int1 := "Unit1.Em7.ControlNodes".cm.softCam.sepaGripperAxisC.waitPos.inPos OR "Unit1.Em7.ControlNodes".cm.softCam.sepaGripperAxisC.ngDischargePos.inPos,
                           intOut := "Unit1.Em7.HmiInterface".intCondition.Actuator_43.intOut,
                           Moveing_INT => "Unit1.Em7.ControlNodes".cm.interlock.stackGripperFwdBwd.work);
   "Unit1.Em7.ControlNodes".cmStackGripperFwdBwd.commands.commandWorkPos := NOT (NOT "Unit1.Em7.ControlNodes".sepaGripper."step".action1[220] AND NOT "Unit1.Em7.ControlNodes".sepaGripper."step".action1[1130]);
END_REGION

REGION Network 269: Call instCmStackGripperFwdBwd (LBC_TwoWayActuator)
   RUNG wire#powerrail
      #instCmStackGripperFwdBwd(enable := TRUE, parentReferenceDesignator := "Unit1.Em7.Config".em.referenceDesignator.combined, feedbackHomePos := "BA030AZSBK22.03", feedbackWorkPos := "BA030AZSBK22.13", enableManualCmds := #statEnableManualCmds, interlockWorkPos := "Unit1.Em7.ControlNodes".cm.interlock.stackGripperFwdBwd.work, interlockHomePos := "Unit1.Em7.ControlNodes".cm.interlock.stackGripperFwdBwd.home, configuration := "Unit1.Em7.Config".cmStackGripperFwdBwd, moduleInterface := "Unit1.Em7.HmiInterface".cmStackGripperFwdBwd, controlNode := "Unit1.Em7.ControlNodes".cmStackGripperFwdBwd, goToHomePos => "BA030AZSPM03.15", goToWorkPos => "BA030AZSPM03.14")
   END_RUNG
   // the same network as SCL:
   #instCmStackGripperFwdBwd(enable := TRUE,   // "LBC_TwoWayActuatorCn"
                           parentReferenceDesignator := "Unit1.Em7.Config".em.referenceDesignator.combined,
                           feedbackHomePos := "BA030AZSBK22.03",
                           feedbackWorkPos := "BA030AZSBK22.13",
                           enableManualCmds := #statEnableManualCmds,
                           interlockWorkPos := "Unit1.Em7.ControlNodes".cm.interlock.stackGripperFwdBwd.work,
                           interlockHomePos := "Unit1.Em7.ControlNodes".cm.interlock.stackGripperFwdBwd.home,
                           configuration := "Unit1.Em7.Config".cmStackGripperFwdBwd,
                           moduleInterface := "Unit1.Em7.HmiInterface".cmStackGripperFwdBwd,
                           controlNode := "Unit1.Em7.ControlNodes".cmStackGripperFwdBwd,
                           goToHomePos => "BA030AZSPM03.15",
                           goToWorkPos => "BA030AZSPM03.14");
END_REGION

REGION Network 271: CmJRWinderClampTopRearUpDown Home
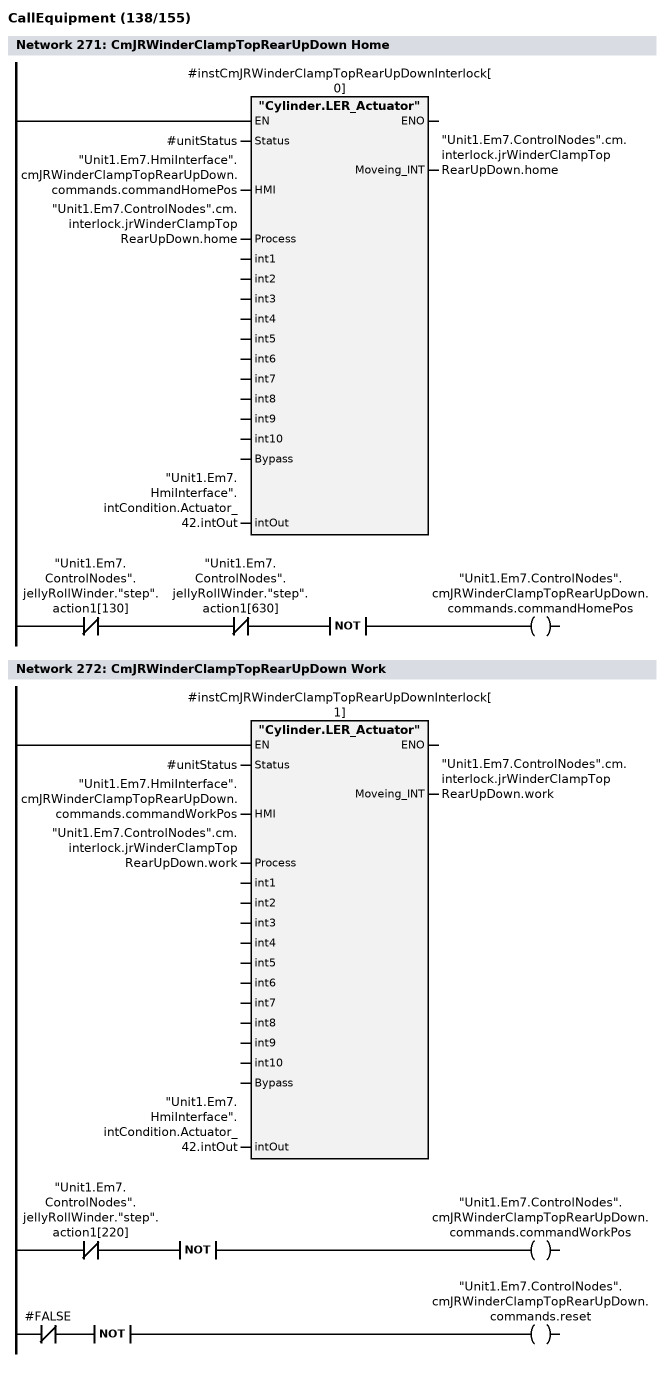
   RUNG wire#powerrail
      #instCmJRWinderClampTopRearUpDownInterlock[0](Status := #unitStatus, HMI := "Unit1.Em7.HmiInterface".cmJRWinderClampTopRearUpDown.commands.commandHomePos, Process := "Unit1.Em7.ControlNodes".cm.interlock.jrWinderClampTopRearUpDown.home, int1 :=, int2 :=, int3 :=, int4 :=, int5 :=, int6 :=, int7 :=, int8 :=, int9 :=, int10 :=, Bypass :=, intOut := "Unit1.Em7.HmiInterface".intCondition.Actuator_42.intOut, Moveing_INT => "Unit1.Em7.ControlNodes".cm.interlock.jrWinderClampTopRearUpDown.home)
   END_RUNG
   RUNG wire#powerrail
      I_Contact( "Unit1.Em7.ControlNodes".jellyRollWinder."step".action1[130] )
      I_Contact( "Unit1.Em7.ControlNodes".jellyRollWinder."step".action1[630] )
      Not()
      Coil( "Unit1.Em7.ControlNodes".cmJRWinderClampTopRearUpDown.commands.commandHomePos )
   END_RUNG
   // the same network as SCL:
   #instCmJRWinderClampTopRearUpDownInterlock[0](Status := #unitStatus,   // "Cylinder.LER_Actuator"
                           HMI := "Unit1.Em7.HmiInterface".cmJRWinderClampTopRearUpDown.commands.commandHomePos,
                           Process := "Unit1.Em7.ControlNodes".cm.interlock.jrWinderClampTopRearUpDown.home,
                           intOut := "Unit1.Em7.HmiInterface".intCondition.Actuator_42.intOut,
                           Moveing_INT => "Unit1.Em7.ControlNodes".cm.interlock.jrWinderClampTopRearUpDown.home);
   "Unit1.Em7.ControlNodes".cmJRWinderClampTopRearUpDown.commands.commandHomePos := NOT (NOT "Unit1.Em7.ControlNodes".jellyRollWinder."step".action1[130] AND NOT "Unit1.Em7.ControlNodes".jellyRollWinder."step".action1[630]);
END_REGION

REGION Network 272: CmJRWinderClampTopRearUpDown Work
   RUNG wire#powerrail
      #instCmJRWinderClampTopRearUpDownInterlock[1](Status := #unitStatus, HMI := "Unit1.Em7.HmiInterface".cmJRWinderClampTopRearUpDown.commands.commandWorkPos, Process := "Unit1.Em7.ControlNodes".cm.interlock.jrWinderClampTopRearUpDown.work, int1 :=, int2 :=, int3 :=, int4 :=, int5 :=, int6 :=, int7 :=, int8 :=, int9 :=, int10 :=, Bypass :=, intOut := "Unit1.Em7.HmiInterface".intCondition.Actuator_42.intOut, Moveing_INT => "Unit1.Em7.ControlNodes".cm.interlock.jrWinderClampTopRearUpDown.work)
   END_RUNG
   RUNG wire#powerrail
      I_Contact( "Unit1.Em7.ControlNodes".jellyRollWinder."step".action1[220] )
      Not()
      Coil( "Unit1.Em7.ControlNodes".cmJRWinderClampTopRearUpDown.commands.commandWorkPos )
   END_RUNG
   RUNG wire#powerrail
      I_Contact( #FALSE )
      Not()
      Coil( "Unit1.Em7.ControlNodes".cmJRWinderClampTopRearUpDown.commands.reset )
   END_RUNG
   // the same network as SCL:
   #instCmJRWinderClampTopRearUpDownInterlock[1](Status := #unitStatus,   // "Cylinder.LER_Actuator"
                           HMI := "Unit1.Em7.HmiInterface".cmJRWinderClampTopRearUpDown.commands.commandWorkPos,
                           Process := "Unit1.Em7.ControlNodes".cm.interlock.jrWinderClampTopRearUpDown.work,
                           intOut := "Unit1.Em7.HmiInterface".intCondition.Actuator_42.intOut,
                           Moveing_INT => "Unit1.Em7.ControlNodes".cm.interlock.jrWinderClampTopRearUpDown.work);
   "Unit1.Em7.ControlNodes".cmJRWinderClampTopRearUpDown.commands.commandWorkPos := NOT (NOT "Unit1.Em7.ControlNodes".jellyRollWinder."step".action1[220]);
   "Unit1.Em7.ControlNodes".cmJRWinderClampTopRearUpDown.commands.reset := NOT (NOT #FALSE);
END_REGION

REGION Network 273: Call instCmJRWinderClampTopRearUpDown (LBC_TwoWayActuator)
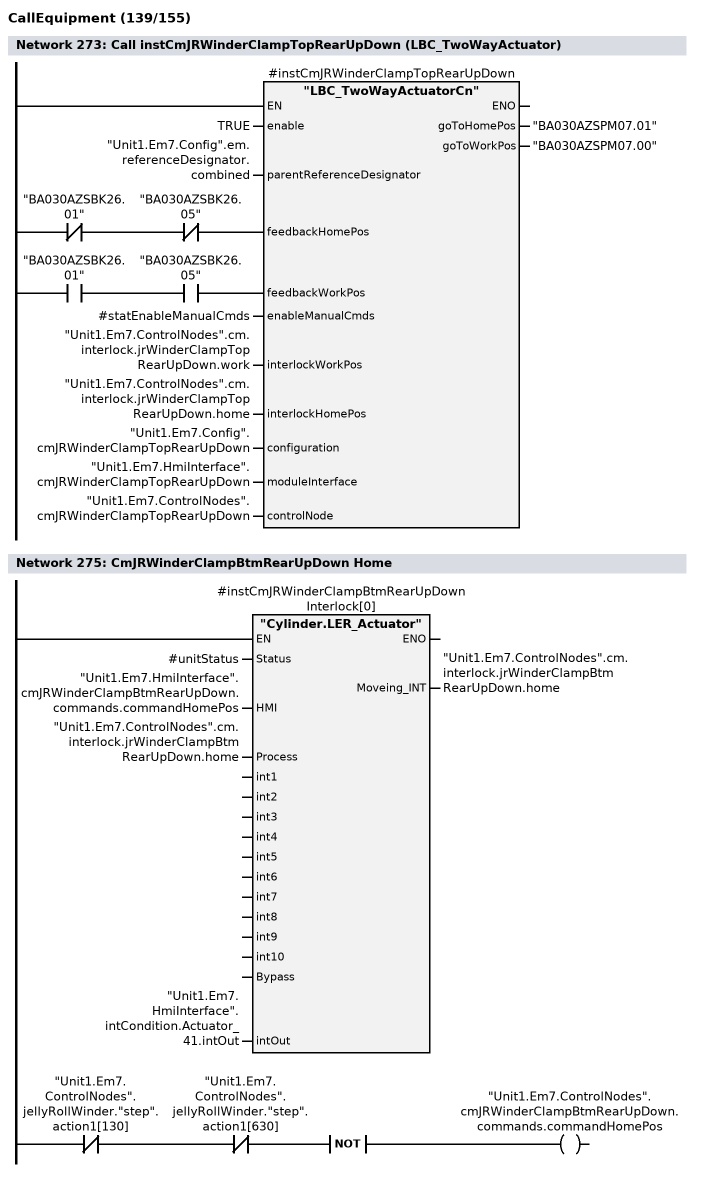
   RUNG wire#powerrail
      #instCmJRWinderClampTopRearUpDown(feedbackHomePos := wire#w1, feedbackWorkPos := wire#w2, enable := TRUE, parentReferenceDesignator := "Unit1.Em7.Config".em.referenceDesignator.combined, enableManualCmds := #statEnableManualCmds, interlockWorkPos := "Unit1.Em7.ControlNodes".cm.interlock.jrWinderClampTopRearUpDown.work, interlockHomePos := "Unit1.Em7.ControlNodes".cm.interlock.jrWinderClampTopRearUpDown.home, configuration := "Unit1.Em7.Config".cmJRWinderClampTopRearUpDown, moduleInterface := "Unit1.Em7.HmiInterface".cmJRWinderClampTopRearUpDown, controlNode := "Unit1.Em7.ControlNodes".cmJRWinderClampTopRearUpDown, goToHomePos => "BA030AZSPM07.01", goToWorkPos => "BA030AZSPM07.00")
   END_RUNG
   RUNG wire#powerrail
      I_Contact( "BA030AZSBK26.01" )
      I_Contact( "BA030AZSBK26.05" )
   END_RUNG wire#w1
   RUNG wire#powerrail
      Contact( "BA030AZSBK26.01" )
      Contact( "BA030AZSBK26.05" )
   END_RUNG wire#w2
   // the same network as SCL:
   #instCmJRWinderClampTopRearUpDown(enable := TRUE,   // "LBC_TwoWayActuatorCn"
                           parentReferenceDesignator := "Unit1.Em7.Config".em.referenceDesignator.combined,
                           feedbackHomePos := NOT "BA030AZSBK26.01" AND NOT "BA030AZSBK26.05",
                           feedbackWorkPos := "BA030AZSBK26.01" AND "BA030AZSBK26.05",
                           enableManualCmds := #statEnableManualCmds,
                           interlockWorkPos := "Unit1.Em7.ControlNodes".cm.interlock.jrWinderClampTopRearUpDown.work,
                           interlockHomePos := "Unit1.Em7.ControlNodes".cm.interlock.jrWinderClampTopRearUpDown.home,
                           configuration := "Unit1.Em7.Config".cmJRWinderClampTopRearUpDown,
                           moduleInterface := "Unit1.Em7.HmiInterface".cmJRWinderClampTopRearUpDown,
                           controlNode := "Unit1.Em7.ControlNodes".cmJRWinderClampTopRearUpDown,
                           goToHomePos => "BA030AZSPM07.01",
                           goToWorkPos => "BA030AZSPM07.00");
END_REGION

REGION Network 275: CmJRWinderClampBtmRearUpDown Home
   RUNG wire#powerrail
      #instCmJRWinderClampBtmRearUpDownInterlock[0](Status := #unitStatus, HMI := "Unit1.Em7.HmiInterface".cmJRWinderClampBtmRearUpDown.commands.commandHomePos, Process := "Unit1.Em7.ControlNodes".cm.interlock.jrWinderClampBtmRearUpDown.home, int1 :=, int2 :=, int3 :=, int4 :=, int5 :=, int6 :=, int7 :=, int8 :=, int9 :=, int10 :=, Bypass :=, intOut := "Unit1.Em7.HmiInterface".intCondition.Actuator_41.intOut, Moveing_INT => "Unit1.Em7.ControlNodes".cm.interlock.jrWinderClampBtmRearUpDown.home)
   END_RUNG
   RUNG wire#powerrail
      I_Contact( "Unit1.Em7.ControlNodes".jellyRollWinder."step".action1[130] )
      I_Contact( "Unit1.Em7.ControlNodes".jellyRollWinder."step".action1[630] )
      Not()
      Coil( "Unit1.Em7.ControlNodes".cmJRWinderClampBtmRearUpDown.commands.commandHomePos )
   END_RUNG
   // the same network as SCL:
   #instCmJRWinderClampBtmRearUpDownInterlock[0](Status := #unitStatus,   // "Cylinder.LER_Actuator"
                           HMI := "Unit1.Em7.HmiInterface".cmJRWinderClampBtmRearUpDown.commands.commandHomePos,
                           Process := "Unit1.Em7.ControlNodes".cm.interlock.jrWinderClampBtmRearUpDown.home,
                           intOut := "Unit1.Em7.HmiInterface".intCondition.Actuator_41.intOut,
                           Moveing_INT => "Unit1.Em7.ControlNodes".cm.interlock.jrWinderClampBtmRearUpDown.home);
   "Unit1.Em7.ControlNodes".cmJRWinderClampBtmRearUpDown.commands.commandHomePos := NOT (NOT "Unit1.Em7.ControlNodes".jellyRollWinder."step".action1[130] AND NOT "Unit1.Em7.ControlNodes".jellyRollWinder."step".action1[630]);
END_REGION

REGION Network 276: CmJRWinderClampBtmRearUpDown Work, Reset
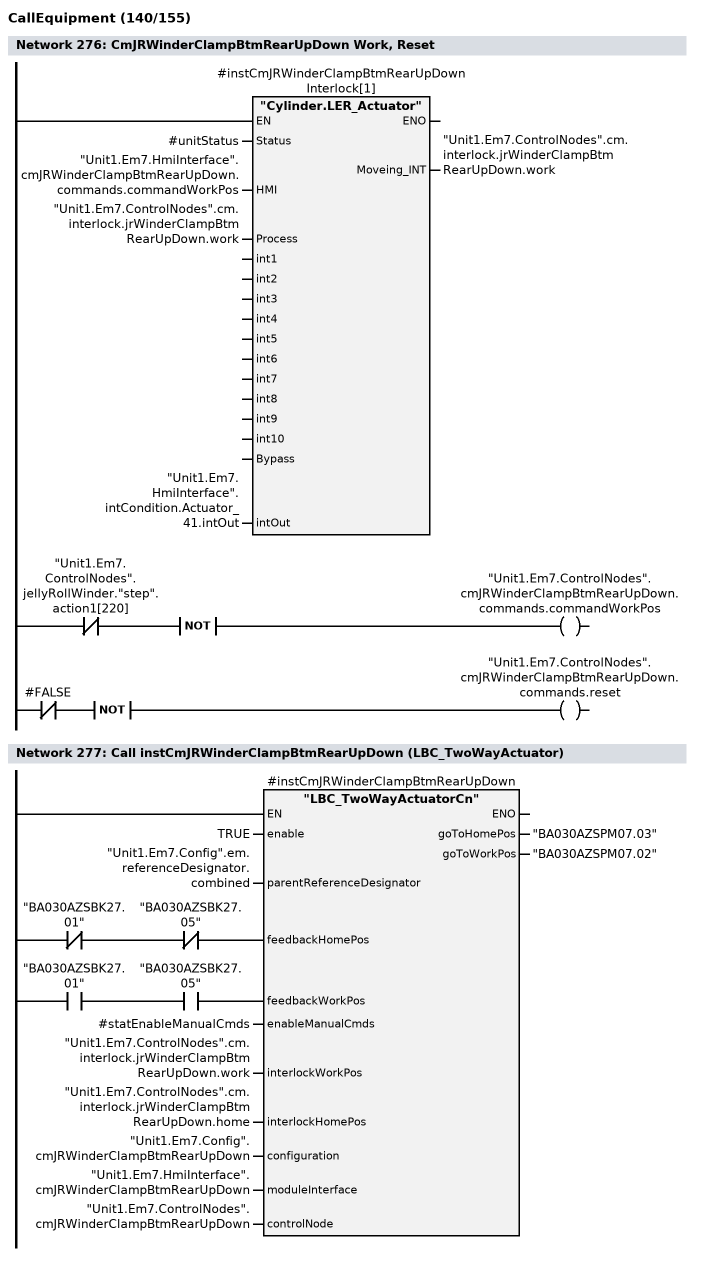
   RUNG wire#powerrail
      #instCmJRWinderClampBtmRearUpDownInterlock[1](Status := #unitStatus, HMI := "Unit1.Em7.HmiInterface".cmJRWinderClampBtmRearUpDown.commands.commandWorkPos, Process := "Unit1.Em7.ControlNodes".cm.interlock.jrWinderClampBtmRearUpDown.work, int1 :=, int2 :=, int3 :=, int4 :=, int5 :=, int6 :=, int7 :=, int8 :=, int9 :=, int10 :=, Bypass :=, intOut := "Unit1.Em7.HmiInterface".intCondition.Actuator_41.intOut, Moveing_INT => "Unit1.Em7.ControlNodes".cm.interlock.jrWinderClampBtmRearUpDown.work)
   END_RUNG
   RUNG wire#powerrail
      I_Contact( "Unit1.Em7.ControlNodes".jellyRollWinder."step".action1[220] )
      Not()
      Coil( "Unit1.Em7.ControlNodes".cmJRWinderClampBtmRearUpDown.commands.commandWorkPos )
   END_RUNG
   RUNG wire#powerrail
      I_Contact( #FALSE )
      Not()
      Coil( "Unit1.Em7.ControlNodes".cmJRWinderClampBtmRearUpDown.commands.reset )
   END_RUNG
   // the same network as SCL:
   #instCmJRWinderClampBtmRearUpDownInterlock[1](Status := #unitStatus,   // "Cylinder.LER_Actuator"
                           HMI := "Unit1.Em7.HmiInterface".cmJRWinderClampBtmRearUpDown.commands.commandWorkPos,
                           Process := "Unit1.Em7.ControlNodes".cm.interlock.jrWinderClampBtmRearUpDown.work,
                           intOut := "Unit1.Em7.HmiInterface".intCondition.Actuator_41.intOut,
                           Moveing_INT => "Unit1.Em7.ControlNodes".cm.interlock.jrWinderClampBtmRearUpDown.work);
   "Unit1.Em7.ControlNodes".cmJRWinderClampBtmRearUpDown.commands.commandWorkPos := NOT (NOT "Unit1.Em7.ControlNodes".jellyRollWinder."step".action1[220]);
   "Unit1.Em7.ControlNodes".cmJRWinderClampBtmRearUpDown.commands.reset := NOT (NOT #FALSE);
END_REGION

REGION Network 277: Call instCmJRWinderClampBtmRearUpDown (LBC_TwoWayActuator)
   RUNG wire#powerrail
      #instCmJRWinderClampBtmRearUpDown(feedbackHomePos := wire#w1, feedbackWorkPos := wire#w2, enable := TRUE, parentReferenceDesignator := "Unit1.Em7.Config".em.referenceDesignator.combined, enableManualCmds := #statEnableManualCmds, interlockWorkPos := "Unit1.Em7.ControlNodes".cm.interlock.jrWinderClampBtmRearUpDown.work, interlockHomePos := "Unit1.Em7.ControlNodes".cm.interlock.jrWinderClampBtmRearUpDown.home, configuration := "Unit1.Em7.Config".cmJRWinderClampBtmRearUpDown, moduleInterface := "Unit1.Em7.HmiInterface".cmJRWinderClampBtmRearUpDown, controlNode := "Unit1.Em7.ControlNodes".cmJRWinderClampBtmRearUpDown, goToHomePos => "BA030AZSPM07.03", goToWorkPos => "BA030AZSPM07.02")
   END_RUNG
   RUNG wire#powerrail
      I_Contact( "BA030AZSBK27.01" )
      I_Contact( "BA030AZSBK27.05" )
   END_RUNG wire#w1
   RUNG wire#powerrail
      Contact( "BA030AZSBK27.01" )
      Contact( "BA030AZSBK27.05" )
   END_RUNG wire#w2
   // the same network as SCL:
   #instCmJRWinderClampBtmRearUpDown(enable := TRUE,   // "LBC_TwoWayActuatorCn"
                           parentReferenceDesignator := "Unit1.Em7.Config".em.referenceDesignator.combined,
                           feedbackHomePos := NOT "BA030AZSBK27.01" AND NOT "BA030AZSBK27.05",
                           feedbackWorkPos := "BA030AZSBK27.01" AND "BA030AZSBK27.05",
                           enableManualCmds := #statEnableManualCmds,
                           interlockWorkPos := "Unit1.Em7.ControlNodes".cm.interlock.jrWinderClampBtmRearUpDown.work,
                           interlockHomePos := "Unit1.Em7.ControlNodes".cm.interlock.jrWinderClampBtmRearUpDown.home,
                           configuration := "Unit1.Em7.Config".cmJRWinderClampBtmRearUpDown,
                           moduleInterface := "Unit1.Em7.HmiInterface".cmJRWinderClampBtmRearUpDown,
                           controlNode := "Unit1.Em7.ControlNodes".cmJRWinderClampBtmRearUpDown,
                           goToHomePos => "BA030AZSPM07.03",
                           goToWorkPos => "BA030AZSPM07.02");
END_REGION

REGION Network 279: CmJRWinderClampTopFrontUpDown Home
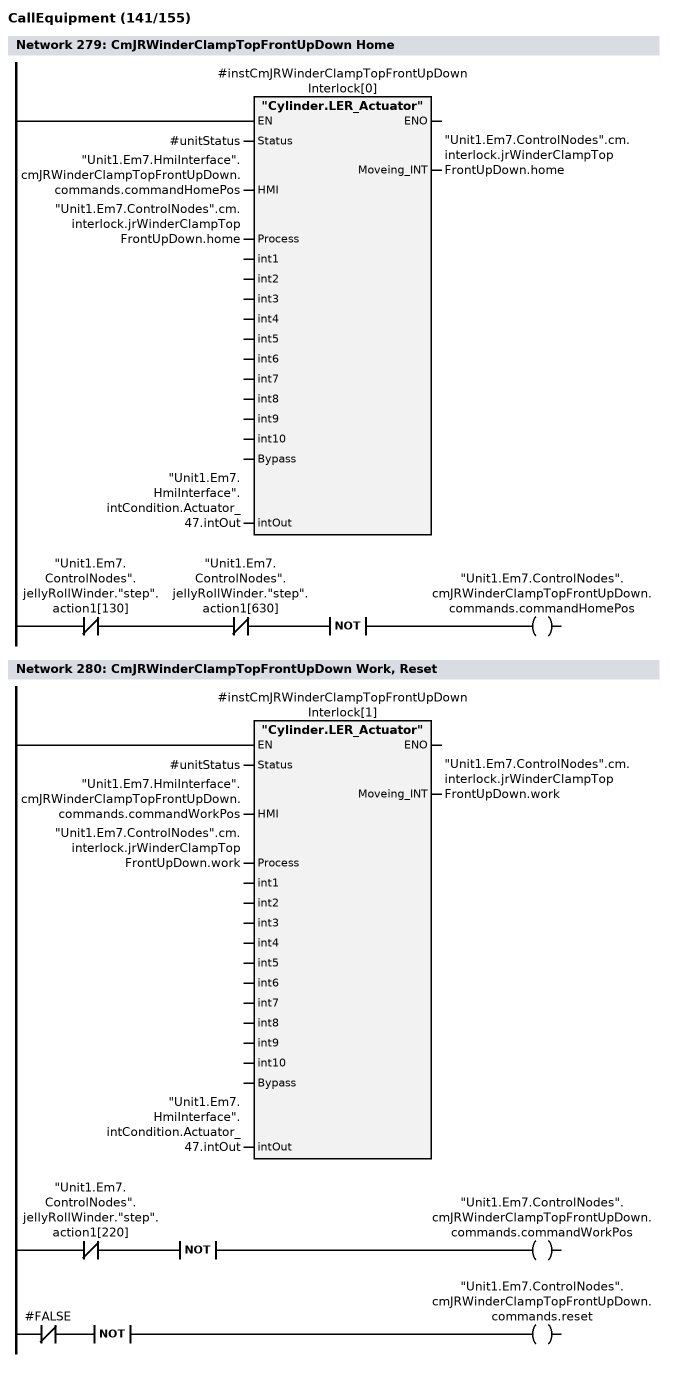
   RUNG wire#powerrail
      #instCmJRWinderClampTopFrontUpDownInterlock[0](Status := #unitStatus, HMI := "Unit1.Em7.HmiInterface".cmJRWinderClampTopFrontUpDown.commands.commandHomePos, Process := "Unit1.Em7.ControlNodes".cm.interlock.jrWinderClampTopFrontUpDown.home, int1 :=, int2 :=, int3 :=, int4 :=, int5 :=, int6 :=, int7 :=, int8 :=, int9 :=, int10 :=, Bypass :=, intOut := "Unit1.Em7.HmiInterface".intCondition.Actuator_47.intOut, Moveing_INT => "Unit1.Em7.ControlNodes".cm.interlock.jrWinderClampTopFrontUpDown.home)
   END_RUNG
   RUNG wire#powerrail
      I_Contact( "Unit1.Em7.ControlNodes".jellyRollWinder."step".action1[130] )
      I_Contact( "Unit1.Em7.ControlNodes".jellyRollWinder."step".action1[630] )
      Not()
      Coil( "Unit1.Em7.ControlNodes".cmJRWinderClampTopFrontUpDown.commands.commandHomePos )
   END_RUNG
   // the same network as SCL:
   #instCmJRWinderClampTopFrontUpDownInterlock[0](Status := #unitStatus,   // "Cylinder.LER_Actuator"
                           HMI := "Unit1.Em7.HmiInterface".cmJRWinderClampTopFrontUpDown.commands.commandHomePos,
                           Process := "Unit1.Em7.ControlNodes".cm.interlock.jrWinderClampTopFrontUpDown.home,
                           intOut := "Unit1.Em7.HmiInterface".intCondition.Actuator_47.intOut,
                           Moveing_INT => "Unit1.Em7.ControlNodes".cm.interlock.jrWinderClampTopFrontUpDown.home);
   "Unit1.Em7.ControlNodes".cmJRWinderClampTopFrontUpDown.commands.commandHomePos := NOT (NOT "Unit1.Em7.ControlNodes".jellyRollWinder."step".action1[130] AND NOT "Unit1.Em7.ControlNodes".jellyRollWinder."step".action1[630]);
END_REGION

REGION Network 280: CmJRWinderClampTopFrontUpDown Work, Reset
   RUNG wire#powerrail
      #instCmJRWinderClampTopFrontUpDownInterlock[1](Status := #unitStatus, HMI := "Unit1.Em7.HmiInterface".cmJRWinderClampTopFrontUpDown.commands.commandWorkPos, Process := "Unit1.Em7.ControlNodes".cm.interlock.jrWinderClampTopFrontUpDown.work, int1 :=, int2 :=, int3 :=, int4 :=, int5 :=, int6 :=, int7 :=, int8 :=, int9 :=, int10 :=, Bypass :=, intOut := "Unit1.Em7.HmiInterface".intCondition.Actuator_47.intOut, Moveing_INT => "Unit1.Em7.ControlNodes".cm.interlock.jrWinderClampTopFrontUpDown.work)
   END_RUNG
   RUNG wire#powerrail
      I_Contact( "Unit1.Em7.ControlNodes".jellyRollWinder."step".action1[220] )
      Not()
      Coil( "Unit1.Em7.ControlNodes".cmJRWinderClampTopFrontUpDown.commands.commandWorkPos )
   END_RUNG
   RUNG wire#powerrail
      I_Contact( #FALSE )
      Not()
      Coil( "Unit1.Em7.ControlNodes".cmJRWinderClampTopFrontUpDown.commands.reset )
   END_RUNG
   // the same network as SCL:
   #instCmJRWinderClampTopFrontUpDownInterlock[1](Status := #unitStatus,   // "Cylinder.LER_Actuator"
                           HMI := "Unit1.Em7.HmiInterface".cmJRWinderClampTopFrontUpDown.commands.commandWorkPos,
                           Process := "Unit1.Em7.ControlNodes".cm.interlock.jrWinderClampTopFrontUpDown.work,
                           intOut := "Unit1.Em7.HmiInterface".intCondition.Actuator_47.intOut,
                           Moveing_INT => "Unit1.Em7.ControlNodes".cm.interlock.jrWinderClampTopFrontUpDown.work);
   "Unit1.Em7.ControlNodes".cmJRWinderClampTopFrontUpDown.commands.commandWorkPos := NOT (NOT "Unit1.Em7.ControlNodes".jellyRollWinder."step".action1[220]);
   "Unit1.Em7.ControlNodes".cmJRWinderClampTopFrontUpDown.commands.reset := NOT (NOT #FALSE);
END_REGION

REGION Network 281: Call instCmJRWinderClampTopFrontUpDown (LBC_TwoWayActuator)
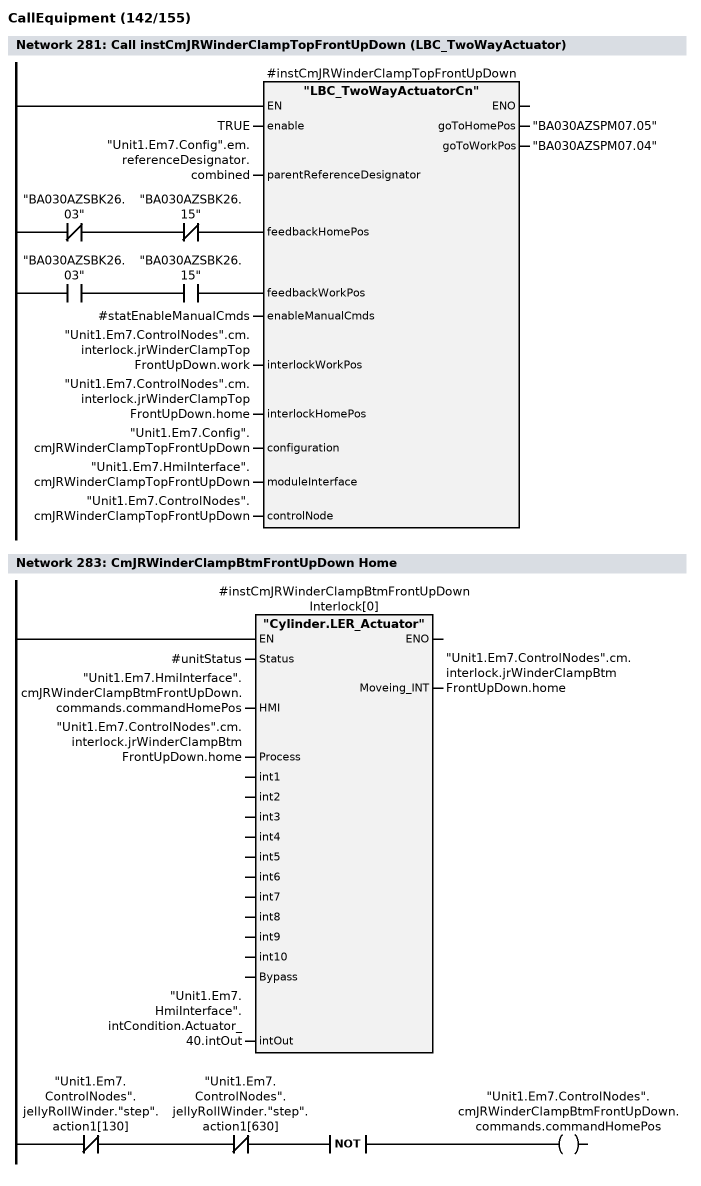
   RUNG wire#powerrail
      #instCmJRWinderClampTopFrontUpDown(feedbackHomePos := wire#w1, feedbackWorkPos := wire#w2, enable := TRUE, parentReferenceDesignator := "Unit1.Em7.Config".em.referenceDesignator.combined, enableManualCmds := #statEnableManualCmds, interlockWorkPos := "Unit1.Em7.ControlNodes".cm.interlock.jrWinderClampTopFrontUpDown.work, interlockHomePos := "Unit1.Em7.ControlNodes".cm.interlock.jrWinderClampTopFrontUpDown.home, configuration := "Unit1.Em7.Config".cmJRWinderClampTopFrontUpDown, moduleInterface := "Unit1.Em7.HmiInterface".cmJRWinderClampTopFrontUpDown, controlNode := "Unit1.Em7.ControlNodes".cmJRWinderClampTopFrontUpDown, goToHomePos => "BA030AZSPM07.05", goToWorkPos => "BA030AZSPM07.04")
   END_RUNG
   RUNG wire#powerrail
      I_Contact( "BA030AZSBK26.03" )
      I_Contact( "BA030AZSBK26.15" )
   END_RUNG wire#w1
   RUNG wire#powerrail
      Contact( "BA030AZSBK26.03" )
      Contact( "BA030AZSBK26.15" )
   END_RUNG wire#w2
   // the same network as SCL:
   #instCmJRWinderClampTopFrontUpDown(enable := TRUE,   // "LBC_TwoWayActuatorCn"
                           parentReferenceDesignator := "Unit1.Em7.Config".em.referenceDesignator.combined,
                           feedbackHomePos := NOT "BA030AZSBK26.03" AND NOT "BA030AZSBK26.15",
                           feedbackWorkPos := "BA030AZSBK26.03" AND "BA030AZSBK26.15",
                           enableManualCmds := #statEnableManualCmds,
                           interlockWorkPos := "Unit1.Em7.ControlNodes".cm.interlock.jrWinderClampTopFrontUpDown.work,
                           interlockHomePos := "Unit1.Em7.ControlNodes".cm.interlock.jrWinderClampTopFrontUpDown.home,
                           configuration := "Unit1.Em7.Config".cmJRWinderClampTopFrontUpDown,
                           moduleInterface := "Unit1.Em7.HmiInterface".cmJRWinderClampTopFrontUpDown,
                           controlNode := "Unit1.Em7.ControlNodes".cmJRWinderClampTopFrontUpDown,
                           goToHomePos => "BA030AZSPM07.05",
                           goToWorkPos => "BA030AZSPM07.04");
END_REGION

REGION Network 283: CmJRWinderClampBtmFrontUpDown Home
   RUNG wire#powerrail
      #instCmJRWinderClampBtmFrontUpDownInterlock[0](Status := #unitStatus, HMI := "Unit1.Em7.HmiInterface".cmJRWinderClampBtmFrontUpDown.commands.commandHomePos, Process := "Unit1.Em7.ControlNodes".cm.interlock.jrWinderClampBtmFrontUpDown.home, int1 :=, int2 :=, int3 :=, int4 :=, int5 :=, int6 :=, int7 :=, int8 :=, int9 :=, int10 :=, Bypass :=, intOut := "Unit1.Em7.HmiInterface".intCondition.Actuator_40.intOut, Moveing_INT => "Unit1.Em7.ControlNodes".cm.interlock.jrWinderClampBtmFrontUpDown.home)
   END_RUNG
   RUNG wire#powerrail
      I_Contact( "Unit1.Em7.ControlNodes".jellyRollWinder."step".action1[130] )
      I_Contact( "Unit1.Em7.ControlNodes".jellyRollWinder."step".action1[630] )
      Not()
      Coil( "Unit1.Em7.ControlNodes".cmJRWinderClampBtmFrontUpDown.commands.commandHomePos )
   END_RUNG
   // the same network as SCL:
   #instCmJRWinderClampBtmFrontUpDownInterlock[0](Status := #unitStatus,   // "Cylinder.LER_Actuator"
                           HMI := "Unit1.Em7.HmiInterface".cmJRWinderClampBtmFrontUpDown.commands.commandHomePos,
                           Process := "Unit1.Em7.ControlNodes".cm.interlock.jrWinderClampBtmFrontUpDown.home,
                           intOut := "Unit1.Em7.HmiInterface".intCondition.Actuator_40.intOut,
                           Moveing_INT => "Unit1.Em7.ControlNodes".cm.interlock.jrWinderClampBtmFrontUpDown.home);
   "Unit1.Em7.ControlNodes".cmJRWinderClampBtmFrontUpDown.commands.commandHomePos := NOT (NOT "Unit1.Em7.ControlNodes".jellyRollWinder."step".action1[130] AND NOT "Unit1.Em7.ControlNodes".jellyRollWinder."step".action1[630]);
END_REGION

REGION Network 284: CmJRWinderClampBtmFrontUpDown Work, Reset
